   S707_WELD_BUFF_DATA8.RBT7_BT_CODE_NO := W#16#0;
   S707_WELD_BUFF_DATA8.RBT7_WELD_COUNT := W#16#0;
   S707_WELD_BUFF_DATA8.RBT8_BT_CODE_NO := W#16#0;
   S707_WELD_BUFF_DATA8.RBT8_WELD_COUNT := W#16#0;
   S707_WELD_BUFF_DATA8.RBT9_BT_CODE_NO := W#16#0;
   S707_WELD_BUFF_DATA8.RBT9_WELD_COUNT := W#16#0;
   S707_WELD_BUFF_DATA8.RBT10_BT_CODE_NO := W#16#0;
   S707_WELD_BUFF_DATA8.RBT10_WELD_COUNT := W#16#0;
   S707_WELD_BUFF_DATA8.RBT11_BT_CODE_NO := W#16#0;
   S707_WELD_BUFF_DATA8.RBT11_WELD_COUNT := W#16#0;
   S707_WELD_BUFF_DATA8.RBT12_BT_CODE_NO := W#16#0;
   S707_WELD_BUFF_DATA8.RBT12_WELD_COUNT := W#16#0;
   S707_WELD_BUFF_DATA8.RBT13_BT_CODE_NO := W#16#0;
   S707_WELD_BUFF_DATA8.RBT13_WELD_COUNT := W#16#0;
   S707_WELD_BUFF_DATA8.RBT14_BT_CODE_NO := W#16#0;
   S707_WELD_BUFF_DATA8.RBT14_WELD_COUNT := W#16#0;
   S707_WELD_BUFF_DATA8.RBT15_BT_CODE_NO := W#16#0;
   S707_WELD_BUFF_DATA8.RBT15_WELD_COUNT := W#16#0;
   S707_WELD_BUFF_DATA8.RBT16_BT_CODE_NO := W#16#0;
   S707_WELD_BUFF_DATA8.RBT16_WELD_COUNT := W#16#0;
   S707_WELD_BUFF_DATA8.RBT17_BT_CODE_NO := W#16#0;
   S707_WELD_BUFF_DATA8.RBT17_WELD_COUNT := W#16#0;
   S707_WELD_BUFF_DATA8.RBT18_BT_CODE_NO := W#16#0;
   S707_WELD_BUFF_DATA8.RBT18_WELD_COUNT := W#16#0;
   S707_WELD_BUFF_DATA8.RBT19_BT_CODE_NO := W#16#0;
   S707_WELD_BUFF_DATA8.RBT19_WELD_COUNT := W#16#0;
   S707_WELD_BUFF_DATA8.RBT20_BT_CODE_NO := W#16#0;
   S707_WELD_BUFF_DATA8.RBT20_WELD_COUNT := W#16#0;
   S707_WELD_BUFF_DATA8.RBT21_BT_CODE_NO := W#16#0;
   S707_WELD_BUFF_DATA8.RBT21_WELD_COUNT := W#16#0;
   S707_WELD_BUFF_DATA8.RBT22_BT_CODE_NO := W#16#0;
   S707_WELD_BUFF_DATA8.RBT22_WELD_COUNT := W#16#0;
   S707_WELD_BUFF_DATA8.RBT23_BT_CODE_NO := W#16#0;
   S707_WELD_BUFF_DATA8.RBT23_WELD_COUNT := W#16#0;
   S707_WELD_BUFF_DATA8.RBT24_BT_CODE_NO := W#16#0;
   S707_WELD_BUFF_DATA8.RBT24_WELD_COUNT := W#16#0;
   S707_WELD_BUFF_DATA8.WELD_DETERMINES_RESULT := W#16#1;
   S707_WELD_BUFF_DATA8.WELD_CHECK_SUM := W#16#3E;
   S707_WELD_BUFF_DATA8.SPARE1 := W#16#0;
   S707_WELD_BUFF_DATA9.STATION_MAIN := W#16#2C3;
   S707_WELD_BUFF_DATA9.DISTINCTION_LH_RH := W#16#1;
   S707_WELD_BUFF_DATA9.STAION_NUMBER := W#16#0;
   S707_WELD_BUFF_DATA9.VIN_NUMBER1 := W#16#0;
   S707_WELD_BUFF_DATA9.VIN_NUMBER2 := W#16#0;
   S707_WELD_BUFF_DATA9.VIN_NUMBER3 := W#16#0;
   S707_WELD_BUFF_DATA9.VIN_NUMBER4 := W#16#2;
   S707_WELD_BUFF_DATA9.SEQ_NUMBER1 := W#16#14;
   S707_WELD_BUFF_DATA9.SEQ_NUMBER2 := W#16#1795;
   S707_WELD_BUFF_DATA9.RBT1_BT_CODE_NO := W#16#835;
   S707_WELD_BUFF_DATA9.RBT1_WELD_COUNT := W#16#F;
   S707_WELD_BUFF_DATA9.RBT2_BT_CODE_NO := W#16#835;
   S707_WELD_BUFF_DATA9.RBT2_WELD_COUNT := W#16#F;
   S707_WELD_BUFF_DATA9.RBT3_BT_CODE_NO := W#16#835;
   S707_WELD_BUFF_DATA9.RBT3_WELD_COUNT := W#16#11;
   S707_WELD_BUFF_DATA9.RBT4_BT_CODE_NO := W#16#835;
   S707_WELD_BUFF_DATA9.RBT4_WELD_COUNT := W#16#F;
   S707_WELD_BUFF_DATA9.RBT5_BT_CODE_NO := W#16#0;
   S707_WELD_BUFF_DATA9.RBT5_WELD_COUNT := W#16#0;
   S707_WELD_BUFF_DATA9.RBT6_BT_CODE_NO := W#16#0;
   S707_WELD_BUFF_DATA9.RBT6_WELD_COUNT := W#16#0;
   S707_WELD_BUFF_DATA9.RBT7_BT_CODE_NO := W#16#0;
   S707_WELD_BUFF_DATA9.RBT7_WELD_COUNT := W#16#0;
   S707_WELD_BUFF_DATA9.RBT8_BT_CODE_NO := W#16#0;
   S707_WELD_BUFF_DATA9.RBT8_WELD_COUNT := W#16#0;
   S707_WELD_BUFF_DATA9.RBT9_BT_CODE_NO := W#16#0;
   S707_WELD_BUFF_DATA9.RBT9_WELD_COUNT := W#16#0;
   S707_WELD_BUFF_DATA9.RBT10_BT_CODE_NO := W#16#0;
   S707_WELD_BUFF_DATA9.RBT10_WELD_COUNT := W#16#0;
   S707_WELD_BUFF_DATA9.RBT11_BT_CODE_NO := W#16#0;
   S707_WELD_BUFF_DATA9.RBT11_WELD_COUNT := W#16#0;
   S707_WELD_BUFF_DATA9.RBT12_BT_CODE_NO := W#16#0;
   S707_WELD_BUFF_DATA9.RBT12_WELD_COUNT := W#16#0;
   S707_WELD_BUFF_DATA9.RBT13_BT_CODE_NO := W#16#0;
   S707_WELD_BUFF_DATA9.RBT13_WELD_COUNT := W#16#0;
   S707_WELD_BUFF_DATA9.RBT14_BT_CODE_NO := W#16#0;
   S707_WELD_BUFF_DATA9.RBT14_WELD_COUNT := W#16#0;
   S707_WELD_BUFF_DATA9.RBT15_BT_CODE_NO := W#16#0;
   S707_WELD_BUFF_DATA9.RBT15_WELD_COUNT := W#16#0;
   S707_WELD_BUFF_DATA9.RBT16_BT_CODE_NO := W#16#0;
   S707_WELD_BUFF_DATA9.RBT16_WELD_COUNT := W#16#0;
   S707_WELD_BUFF_DATA9.RBT17_BT_CODE_NO := W#16#0;
   S707_WELD_BUFF_DATA9.RBT17_WELD_COUNT := W#16#0;
   S707_WELD_BUFF_DATA9.RBT18_BT_CODE_NO := W#16#0;
   S707_WELD_BUFF_DATA9.RBT18_WELD_COUNT := W#16#0;
   S707_WELD_BUFF_DATA9.RBT19_BT_CODE_NO := W#16#0;
   S707_WELD_BUFF_DATA9.RBT19_WELD_COUNT := W#16#0;
   S707_WELD_BUFF_DATA9.RBT20_BT_CODE_NO := W#16#0;
   S707_WELD_BUFF_DATA9.RBT20_WELD_COUNT := W#16#0;
   S707_WELD_BUFF_DATA9.RBT21_BT_CODE_NO := W#16#0;
   S707_WELD_BUFF_DATA9.RBT21_WELD_COUNT := W#16#0;
   S707_WELD_BUFF_DATA9.RBT22_BT_CODE_NO := W#16#0;
   S707_WELD_BUFF_DATA9.RBT22_WELD_COUNT := W#16#0;
   S707_WELD_BUFF_DATA9.RBT23_BT_CODE_NO := W#16#0;
   S707_WELD_BUFF_DATA9.RBT23_WELD_COUNT := W#16#0;
   S707_WELD_BUFF_DATA9.RBT24_BT_CODE_NO := W#16#0;
   S707_WELD_BUFF_DATA9.RBT24_WELD_COUNT := W#16#0;
   S707_WELD_BUFF_DATA9.WELD_DETERMINES_RESULT := W#16#1;
   S707_WELD_BUFF_DATA9.WELD_CHECK_SUM := W#16#3E;
   S707_WELD_BUFF_DATA9.SPARE1 := W#16#0;
   S707_WELD_BUFF_DATA10.STATION_MAIN := W#16#2C3;
   S707_WELD_BUFF_DATA10.DISTINCTION_LH_RH := W#16#1;
   S707_WELD_BUFF_DATA10.STAION_NUMBER := W#16#0;
   S707_WELD_BUFF_DATA10.VIN_NUMBER1 := W#16#0;
   S707_WELD_BUFF_DATA10.VIN_NUMBER2 := W#16#0;
   S707_WELD_BUFF_DATA10.VIN_NUMBER3 := W#16#0;
   S707_WELD_BUFF_DATA10.VIN_NUMBER4 := W#16#2;
   S707_WELD_BUFF_DATA10.SEQ_NUMBER1 := W#16#14;
   S707_WELD_BUFF_DATA10.SEQ_NUMBER2 := W#16#1794;
   S707_WELD_BUFF_DATA10.RBT1_BT_CODE_NO := W#16#835;
   S707_WELD_BUFF_DATA10.RBT1_WELD_COUNT := W#16#F;
   S707_WELD_BUFF_DATA10.RBT2_BT_CODE_NO := W#16#835;
   S707_WELD_BUFF_DATA10.RBT2_WELD_COUNT := W#16#F;
   S707_WELD_BUFF_DATA10.RBT3_BT_CODE_NO := W#16#835;
   S707_WELD_BUFF_DATA10.RBT3_WELD_COUNT := W#16#11;
   S707_WELD_BUFF_DATA10.RBT4_BT_CODE_NO := W#16#835;
   S707_WELD_BUFF_DATA10.RBT4_WELD_COUNT := W#16#F;
   S707_WELD_BUFF_DATA10.RBT5_BT_CODE_NO := W#16#0;
   S707_WELD_BUFF_DATA10.RBT5_WELD_COUNT := W#16#0;
   S707_WELD_BUFF_DATA10.RBT6_BT_CODE_NO := W#16#0;
   S707_WELD_BUFF_DATA10.RBT6_WELD_COUNT := W#16#0;
   S707_WELD_BUFF_DATA10.RBT7_BT_CODE_NO := W#16#0;
   S707_WELD_BUFF_DATA10.RBT7_WELD_COUNT := W#16#0;
   S707_WELD_BUFF_DATA10.RBT8_BT_CODE_NO := W#16#0;
   S707_WELD_BUFF_DATA10.RBT8_WELD_COUNT := W#16#0;
   S707_WELD_BUFF_DATA10.RBT9_BT_CODE_NO := W#16#0;
   S707_WELD_BUFF_DATA10.RBT9_WELD_COUNT := W#16#0;
   S707_WELD_BUFF_DATA10.RBT10_BT_CODE_NO := W#16#0;
   S707_WELD_BUFF_DATA10.RBT10_WELD_COUNT := W#16#0;
   S707_WELD_BUFF_DATA10.RBT11_BT_CODE_NO := W#16#0;
   S707_WELD_BUFF_DATA10.RBT11_WELD_COUNT := W#16#0;
   S707_WELD_BUFF_DATA10.RBT12_BT_CODE_NO := W#16#0;
   S707_WELD_BUFF_DATA10.RBT12_WELD_COUNT := W#16#0;
   S707_WELD_BUFF_DATA10.RBT13_BT_CODE_NO := W#16#0;
   S707_WELD_BUFF_DATA10.RBT13_WELD_COUNT := W#16#0;
   S707_WELD_BUFF_DATA10.RBT14_BT_CODE_NO := W#16#0;
   S707_WELD_BUFF_DATA10.RBT14_WELD_COUNT := W#16#0;
   S707_WELD_BUFF_DATA10.RBT15_BT_CODE_NO := W#16#0;
   S707_WELD_BUFF_DATA10.RBT15_WELD_COUNT := W#16#0;
   S707_WELD_BUFF_DATA10.RBT16_BT_CODE_NO := W#16#0;
   S707_WELD_BUFF_DATA10.RBT16_WELD_COUNT := W#16#0;
   S707_WELD_BUFF_DATA10.RBT17_BT_CODE_NO := W#16#0;
   S707_WELD_BUFF_DATA10.RBT17_WELD_COUNT := W#16#0;
   S707_WELD_BUFF_DATA10.RBT18_BT_CODE_NO := W#16#0;
   S707_WELD_BUFF_DATA10.RBT18_WELD_COUNT := W#16#0;
   S707_WELD_BUFF_DATA10.RBT19_BT_CODE_NO := W#16#0;
   S707_WELD_BUFF_DATA10.RBT19_WELD_COUNT := W#16#0;
   S707_WELD_BUFF_DATA10.RBT20_BT_CODE_NO := W#16#0;
   S707_WELD_BUFF_DATA10.RBT20_WELD_COUNT := W#16#0;
   S707_WELD_BUFF_DATA10.RBT21_BT_CODE_NO := W#16#0;
   S707_WELD_BUFF_DATA10.RBT21_WELD_COUNT := W#16#0;
   S707_WELD_BUFF_DATA10.RBT22_BT_CODE_NO := W#16#0;
   S707_WELD_BUFF_DATA10.RBT22_WELD_COUNT := W#16#0;
   S707_WELD_BUFF_DATA10.RBT23_BT_CODE_NO := W#16#0;
   S707_WELD_BUFF_DATA10.RBT23_WELD_COUNT := W#16#0;
   S707_WELD_BUFF_DATA10.RBT24_BT_CODE_NO := W#16#0;
   S707_WELD_BUFF_DATA10.RBT24_WELD_COUNT := W#16#0;
   S707_WELD_BUFF_DATA10.WELD_DETERMINES_RESULT := W#16#1;
   S707_WELD_BUFF_DATA10.WELD_CHECK_SUM := W#16#3E;
   S707_WELD_BUFF_DATA10.SPARE1 := W#16#0;
   S707_WELD_BUFF_DATA11.STATION_MAIN := W#16#0;
   S707_WELD_BUFF_DATA11.DISTINCTION_LH_RH := W#16#0;
   S707_WELD_BUFF_DATA11.STAION_NUMBER := W#16#0;
   S707_WELD_BUFF_DATA11.VIN_NUMBER1 := W#16#0;
   S707_WELD_BUFF_DATA11.VIN_NUMBER2 := W#16#0;
   S707_WELD_BUFF_DATA11.VIN_NUMBER3 := W#16#0;
   S707_WELD_BUFF_DATA11.VIN_NUMBER4 := W#16#0;
   S707_WELD_BUFF_DATA11.SEQ_NUMBER1 := W#16#0;
   S707_WELD_BUFF_DATA11.SEQ_NUMBER2 := W#16#0;
   S707_WELD_BUFF_DATA11.RBT1_BT_CODE_NO := W#16#0;
   S707_WELD_BUFF_DATA11.RBT1_WELD_COUNT := W#16#0;
   S707_WELD_BUFF_DATA11.RBT2_BT_CODE_NO := W#16#0;
   S707_WELD_BUFF_DATA11.RBT2_WELD_COUNT := W#16#0;
   S707_WELD_BUFF_DATA11.RBT3_BT_CODE_NO := W#16#0;
   S707_WELD_BUFF_DATA11.RBT3_WELD_COUNT := W#16#0;
   S707_WELD_BUFF_DATA11.RBT4_BT_CODE_NO := W#16#0;
   S707_WELD_BUFF_DATA11.RBT4_WELD_COUNT := W#16#0;
   S707_WELD_BUFF_DATA11.RBT5_BT_CODE_NO := W#16#0;
   S707_WELD_BUFF_DATA11.RBT5_WELD_COUNT := W#16#0;
   S707_WELD_BUFF_DATA11.RBT6_BT_CODE_NO := W#16#0;
   S707_WELD_BUFF_DATA11.RBT6_WELD_COUNT := W#16#0;
   S707_WELD_BUFF_DATA11.RBT7_BT_CODE_NO := W#16#0;
   S707_WELD_BUFF_DATA11.RBT7_WELD_COUNT := W#16#0;
   S707_WELD_BUFF_DATA11.RBT8_BT_CODE_NO := W#16#0;
   S707_WELD_BUFF_DATA11.RBT8_WELD_COUNT := W#16#0;
   S707_WELD_BUFF_DATA11.RBT9_BT_CODE_NO := W#16#0;
   S707_WELD_BUFF_DATA11.RBT9_WELD_COUNT := W#16#0;
   S707_WELD_BUFF_DATA11.RBT10_BT_CODE_NO := W#16#0;
   S707_WELD_BUFF_DATA11.RBT10_WELD_COUNT := W#16#0;
   S707_WELD_BUFF_DATA11.RBT11_BT_CODE_NO := W#16#0;
   S707_WELD_BUFF_DATA11.RBT11_WELD_COUNT := W#16#0;
   S707_WELD_BUFF_DATA11.RBT12_BT_CODE_NO := W#16#0;
   S707_WELD_BUFF_DATA11.RBT12_WELD_COUNT := W#16#0;
   S707_WELD_BUFF_DATA11.RBT13_BT_CODE_NO := W#16#0;
   S707_WELD_BUFF_DATA11.RBT13_WELD_COUNT := W#16#0;
   S707_WELD_BUFF_DATA11.RBT14_BT_CODE_NO := W#16#0;
   S707_WELD_BUFF_DATA11.RBT14_WELD_COUNT := W#16#0;
   S707_WELD_BUFF_DATA11.RBT15_BT_CODE_NO := W#16#0;
   S707_WELD_BUFF_DATA11.RBT15_WELD_COUNT := W#16#0;
   S707_WELD_BUFF_DATA11.RBT16_BT_CODE_NO := W#16#0;
   S707_WELD_BUFF_DATA11.RBT16_WELD_COUNT := W#16#0;
   S707_WELD_BUFF_DATA11.RBT17_BT_CODE_NO := W#16#0;
   S707_WELD_BUFF_DATA11.RBT17_WELD_COUNT := W#16#0;
   S707_WELD_BUFF_DATA11.RBT18_BT_CODE_NO := W#16#0;
   S707_WELD_BUFF_DATA11.RBT18_WELD_COUNT := W#16#0;
   S707_WELD_BUFF_DATA11.RBT19_BT_CODE_NO := W#16#0;
   S707_WELD_BUFF_DATA11.RBT19_WELD_COUNT := W#16#0;
   S707_WELD_BUFF_DATA11.RBT20_BT_CODE_NO := W#16#0;
   S707_WELD_BUFF_DATA11.RBT20_WELD_COUNT := W#16#0;
   S707_WELD_BUFF_DATA11.RBT21_BT_CODE_NO := W#16#0;
   S707_WELD_BUFF_DATA11.RBT21_WELD_COUNT := W#16#0;
   S707_WELD_BUFF_DATA11.RBT22_BT_CODE_NO := W#16#0;
   S707_WELD_BUFF_DATA11.RBT22_WELD_COUNT := W#16#0;
   S707_WELD_BUFF_DATA11.RBT23_BT_CODE_NO := W#16#0;
   S707_WELD_BUFF_DATA11.RBT23_WELD_COUNT := W#16#0;
   S707_WELD_BUFF_DATA11.RBT24_BT_CODE_NO := W#16#0;
   S707_WELD_BUFF_DATA11.RBT24_WELD_COUNT := W#16#0;
   S707_WELD_BUFF_DATA11.WELD_DETERMINES_RESULT := W#16#0;
   S707_WELD_BUFF_DATA11.WELD_CHECK_SUM := W#16#0;
   S707_WELD_BUFF_DATA11.SPARE1 := W#16#0;
   S707_WELD_BUFF_DATA21.STATION_MAIN := W#16#0;
   S707_WELD_BUFF_DATA21.DISTINCTION_LH_RH := W#16#0;
   S707_WELD_BUFF_DATA21.STAION_NUMBER := W#16#0;
   S707_WELD_BUFF_DATA21.VIN_NUMBER1 := W#16#0;
   S707_WELD_BUFF_DATA21.VIN_NUMBER2 := W#16#0;
   S707_WELD_BUFF_DATA21.VIN_NUMBER3 := W#16#0;
   S707_WELD_BUFF_DATA21.VIN_NUMBER4 := W#16#0;
   S707_WELD_BUFF_DATA21.SEQ_NUMBER1 := W#16#0;
   S707_WELD_BUFF_DATA21.SEQ_NUMBER2 := W#16#0;
   S707_WELD_BUFF_DATA21.RBT1_BT_CODE_NO := W#16#0;
   S707_WELD_BUFF_DATA21.RBT1_WELD_COUNT := W#16#0;
   S707_WELD_BUFF_DATA21.RBT2_BT_CODE_NO := W#16#0;
   S707_WELD_BUFF_DATA21.RBT2_WELD_COUNT := W#16#0;
   S707_WELD_BUFF_DATA21.RBT3_BT_CODE_NO := W#16#0;
   S707_WELD_BUFF_DATA21.RBT3_WELD_COUNT := W#16#0;
   S707_WELD_BUFF_DATA21.RBT4_BT_CODE_NO := W#16#0;
   S707_WELD_BUFF_DATA21.RBT4_WELD_COUNT := W#16#0;
   S707_WELD_BUFF_DATA21.RBT5_BT_CODE_NO := W#16#0;
   S707_WELD_BUFF_DATA21.RBT5_WELD_COUNT := W#16#0;
   S707_WELD_BUFF_DATA21.RBT6_BT_CODE_NO := W#16#0;
   S707_WELD_BUFF_DATA21.RBT6_WELD_COUNT := W#16#0;
   S707_WELD_BUFF_DATA21.RBT7_BT_CODE_NO := W#16#0;
   S707_WELD_BUFF_DATA21.RBT7_WELD_COUNT := W#16#0;
   S707_WELD_BUFF_DATA21.RBT8_BT_CODE_NO := W#16#0;
   S707_WELD_BUFF_DATA21.RBT8_WELD_COUNT := W#16#0;
   S707_WELD_BUFF_DATA21.RBT9_BT_CODE_NO := W#16#0;
   S707_WELD_BUFF_DATA21.RBT9_WELD_COUNT := W#16#0;
   S707_WELD_BUFF_DATA21.RBT10_BT_CODE_NO := W#16#0;
   S707_WELD_BUFF_DATA21.RBT10_WELD_COUNT := W#16#0;
   S707_WELD_BUFF_DATA21.RBT11_BT_CODE_NO := W#16#0;
   S707_WELD_BUFF_DATA21.RBT11_WELD_COUNT := W#16#0;
   S707_WELD_BUFF_DATA21.RBT12_BT_CODE_NO := W#16#0;
   S707_WELD_BUFF_DATA21.RBT12_WELD_COUNT := W#16#0;
   S707_WELD_BUFF_DATA21.RBT13_BT_CODE_NO := W#16#0;
   S707_WELD_BUFF_DATA21.RBT13_WELD_COUNT := W#16#0;
   S707_WELD_BUFF_DATA21.RBT14_BT_CODE_NO := W#16#0;
   S707_WELD_BUFF_DATA21.RBT14_WELD_COUNT := W#16#0;
   S707_WELD_BUFF_DATA21.RBT15_BT_CODE_NO := W#16#0;
   S707_WELD_BUFF_DATA21.RBT15_WELD_COUNT := W#16#0;
   S707_WELD_BUFF_DATA21.RBT16_BT_CODE_NO := W#16#0;
   S707_WELD_BUFF_DATA21.RBT16_WELD_COUNT := W#16#0;
   S707_WELD_BUFF_DATA21.RBT17_BT_CODE_NO := W#16#0;
   S707_WELD_BUFF_DATA21.RBT17_WELD_COUNT := W#16#0;
   S707_WELD_BUFF_DATA21.RBT18_BT_CODE_NO := W#16#0;
   S707_WELD_BUFF_DATA21.RBT18_WELD_COUNT := W#16#0;
   S707_WELD_BUFF_DATA21.RBT19_BT_CODE_NO := W#16#0;
   S707_WELD_BUFF_DATA21.RBT19_WELD_COUNT := W#16#0;
   S707_WELD_BUFF_DATA21.RBT20_BT_CODE_NO := W#16#0;
   S707_WELD_BUFF_DATA21.RBT20_WELD_COUNT := W#16#0;
   S707_WELD_BUFF_DATA21.RBT21_BT_CODE_NO := W#16#0;
   S707_WELD_BUFF_DATA21.RBT21_WELD_COUNT := W#16#0;
   S707_WELD_BUFF_DATA21.RBT22_BT_CODE_NO := W#16#0;
   S707_WELD_BUFF_DATA21.RBT22_WELD_COUNT := W#16#0;
   S707_WELD_BUFF_DATA21.RBT23_BT_CODE_NO := W#16#0;
   S707_WELD_BUFF_DATA21.RBT23_WELD_COUNT := W#16#0;
   S707_WELD_BUFF_DATA21.RBT24_BT_CODE_NO := W#16#0;
   S707_WELD_BUFF_DATA21.RBT24_WELD_COUNT := W#16#0;
   S707_WELD_BUFF_DATA21.WELD_DETERMINES_RESULT := W#16#0;
   S707_WELD_BUFF_DATA21.WELD_CHECK_SUM := W#16#0;
   S707_WELD_BUFF_DATA21.SPARE1 := W#16#0;
   S707_WELD_BUFF_DATA31.STATION_MAIN := W#16#0;
   S707_WELD_BUFF_DATA31.DISTINCTION_LH_RH := W#16#0;
   S707_WELD_BUFF_DATA31.STAION_NUMBER := W#16#0;
   S707_WELD_BUFF_DATA31.VIN_NUMBER1 := W#16#0;
   S707_WELD_BUFF_DATA31.VIN_NUMBER2 := W#16#0;
   S707_WELD_BUFF_DATA31.VIN_NUMBER3 := W#16#0;
   S707_WELD_BUFF_DATA31.VIN_NUMBER4 := W#16#0;
   S707_WELD_BUFF_DATA31.SEQ_NUMBER1 := W#16#0;
   S707_WELD_BUFF_DATA31.SEQ_NUMBER2 := W#16#0;
   S707_WELD_BUFF_DATA31.RBT1_BT_CODE_NO := W#16#0;
   S707_WELD_BUFF_DATA31.RBT1_WELD_COUNT := W#16#0;
   S707_WELD_BUFF_DATA31.RBT2_BT_CODE_NO := W#16#0;
   S707_WELD_BUFF_DATA31.RBT2_WELD_COUNT := W#16#0;
   S707_WELD_BUFF_DATA31.RBT3_BT_CODE_NO := W#16#0;
   S707_WELD_BUFF_DATA31.RBT3_WELD_COUNT := W#16#0;
   S707_WELD_BUFF_DATA31.RBT4_BT_CODE_NO := W#16#0;
   S707_WELD_BUFF_DATA31.RBT4_WELD_COUNT := W#16#0;
   S707_WELD_BUFF_DATA31.RBT5_BT_CODE_NO := W#16#0;
   S707_WELD_BUFF_DATA31.RBT5_WELD_COUNT := W#16#0;
   S707_WELD_BUFF_DATA31.RBT6_BT_CODE_NO := W#16#0;
   S707_WELD_BUFF_DATA31.RBT6_WELD_COUNT := W#16#0;
   S707_WELD_BUFF_DATA31.RBT7_BT_CODE_NO := W#16#0;
   S707_WELD_BUFF_DATA31.RBT7_WELD_COUNT := W#16#0;
   S707_WELD_BUFF_DATA31.RBT8_BT_CODE_NO := W#16#0;
   S707_WELD_BUFF_DATA31.RBT8_WELD_COUNT := W#16#0;
   S707_WELD_BUFF_DATA31.RBT9_BT_CODE_NO := W#16#0;
   S707_WELD_BUFF_DATA31.RBT9_WELD_COUNT := W#16#0;
   S707_WELD_BUFF_DATA31.RBT10_BT_CODE_NO := W#16#0;
   S707_WELD_BUFF_DATA31.RBT10_WELD_COUNT := W#16#0;
   S707_WELD_BUFF_DATA31.RBT11_BT_CODE_NO := W#16#0;
   S707_WELD_BUFF_DATA31.RBT11_WELD_COUNT := W#16#0;
   S707_WELD_BUFF_DATA31.RBT12_BT_CODE_NO := W#16#0;
   S707_WELD_BUFF_DATA31.RBT12_WELD_COUNT := W#16#0;
   S707_WELD_BUFF_DATA31.RBT13_BT_CODE_NO := W#16#0;
   S707_WELD_BUFF_DATA31.RBT13_WELD_COUNT := W#16#0;
   S707_WELD_BUFF_DATA31.RBT14_BT_CODE_NO := W#16#0;
   S707_WELD_BUFF_DATA31.RBT14_WELD_COUNT := W#16#0;
   S707_WELD_BUFF_DATA31.RBT15_BT_CODE_NO := W#16#0;
   S707_WELD_BUFF_DATA31.RBT15_WELD_COUNT := W#16#0;
   S707_WELD_BUFF_DATA31.RBT16_BT_CODE_NO := W#16#0;
   S707_WELD_BUFF_DATA31.RBT16_WELD_COUNT := W#16#0;
   S707_WELD_BUFF_DATA31.RBT17_BT_CODE_NO := W#16#0;
   S707_WELD_BUFF_DATA31.RBT17_WELD_COUNT := W#16#0;
   S707_WELD_BUFF_DATA31.RBT18_BT_CODE_NO := W#16#0;
   S707_WELD_BUFF_DATA31.RBT18_WELD_COUNT := W#16#0;
   S707_WELD_BUFF_DATA31.RBT19_BT_CODE_NO := W#16#0;
   S707_WELD_BUFF_DATA31.RBT19_WELD_COUNT := W#16#0;
   S707_WELD_BUFF_DATA31.RBT20_BT_CODE_NO := W#16#0;
   S707_WELD_BUFF_DATA31.RBT20_WELD_COUNT := W#16#0;
   S707_WELD_BUFF_DATA31.RBT21_BT_CODE_NO := W#16#0;
   S707_WELD_BUFF_DATA31.RBT21_WELD_COUNT := W#16#0;
   S707_WELD_BUFF_DATA31.RBT22_BT_CODE_NO := W#16#0;
   S707_WELD_BUFF_DATA31.RBT22_WELD_COUNT := W#16#0;
   S707_WELD_BUFF_DATA31.RBT23_BT_CODE_NO := W#16#0;
   S707_WELD_BUFF_DATA31.RBT23_WELD_COUNT := W#16#0;
   S707_WELD_BUFF_DATA31.RBT24_BT_CODE_NO := W#16#0;
   S707_WELD_BUFF_DATA31.RBT24_WELD_COUNT := W#16#0;
   S707_WELD_BUFF_DATA31.WELD_DETERMINES_RESULT := W#16#0;
   S707_WELD_BUFF_DATA31.WELD_CHECK_SUM := W#16#0;
   S707_WELD_BUFF_DATA31.SPARE1 := W#16#0;
   S707_WELD_BUFF_DATA41.STATION_MAIN := W#16#0;
   S707_WELD_BUFF_DATA41.DISTINCTION_LH_RH := W#16#0;
   S707_WELD_BUFF_DATA41.STAION_NUMBER := W#16#0;
   S707_WELD_BUFF_DATA41.VIN_NUMBER1 := W#16#0;
   S707_WELD_BUFF_DATA41.VIN_NUMBER2 := W#16#0;
   S707_WELD_BUFF_DATA41.VIN_NUMBER3 := W#16#0;
   S707_WELD_BUFF_DATA41.VIN_NUMBER4 := W#16#0;
   S707_WELD_BUFF_DATA41.SEQ_NUMBER1 := W#16#0;
   S707_WELD_BUFF_DATA41.SEQ_NUMBER2 := W#16#0;
   S707_WELD_BUFF_DATA41.RBT1_BT_CODE_NO := W#16#0;
   S707_WELD_BUFF_DATA41.RBT1_WELD_COUNT := W#16#0;
   S707_WELD_BUFF_DATA41.RBT2_BT_CODE_NO := W#16#0;
   S707_WELD_BUFF_DATA41.RBT2_WELD_COUNT := W#16#0;
   S707_WELD_BUFF_DATA41.RBT3_BT_CODE_NO := W#16#0;
   S707_WELD_BUFF_DATA41.RBT3_WELD_COUNT := W#16#0;
   S707_WELD_BUFF_DATA41.RBT4_BT_CODE_NO := W#16#0;
   S707_WELD_BUFF_DATA41.RBT4_WELD_COUNT := W#16#0;
   S707_WELD_BUFF_DATA41.RBT5_BT_CODE_NO := W#16#0;
   S707_WELD_BUFF_DATA41.RBT5_WELD_COUNT := W#16#0;
   S707_WELD_BUFF_DATA41.RBT6_BT_CODE_NO := W#16#0;
   S707_WELD_BUFF_DATA41.RBT6_WELD_COUNT := W#16#0;
   S707_WELD_BUFF_DATA41.RBT7_BT_CODE_NO := W#16#0;
   S707_WELD_BUFF_DATA41.RBT7_WELD_COUNT := W#16#0;
   S707_WELD_BUFF_DATA41.RBT8_BT_CODE_NO := W#16#0;
   S707_WELD_BUFF_DATA41.RBT8_WELD_COUNT := W#16#0;
   S707_WELD_BUFF_DATA41.RBT9_BT_CODE_NO := W#16#0;
   S707_WELD_BUFF_DATA41.RBT9_WELD_COUNT := W#16#0;
   S707_WELD_BUFF_DATA41.RBT10_BT_CODE_NO := W#16#0;
   S707_WELD_BUFF_DATA41.RBT10_WELD_COUNT := W#16#0;
   S707_WELD_BUFF_DATA41.RBT11_BT_CODE_NO := W#16#0;
   S707_WELD_BUFF_DATA41.RBT11_WELD_COUNT := W#16#0;
   S707_WELD_BUFF_DATA41.RBT12_BT_CODE_NO := W#16#0;
   S707_WELD_BUFF_DATA41.RBT12_WELD_COUNT := W#16#0;
   S707_WELD_BUFF_DATA41.RBT13_BT_CODE_NO := W#16#0;
   S707_WELD_BUFF_DATA41.RBT13_WELD_COUNT := W#16#0;
   S707_WELD_BUFF_DATA41.RBT14_BT_CODE_NO := W#16#0;
   S707_WELD_BUFF_DATA41.RBT14_WELD_COUNT := W#16#0;
   S707_WELD_BUFF_DATA41.RBT15_BT_CODE_NO := W#16#0;
   S707_WELD_BUFF_DATA41.RBT15_WELD_COUNT := W#16#0;
   S707_WELD_BUFF_DATA41.RBT16_BT_CODE_NO := W#16#0;
   S707_WELD_BUFF_DATA41.RBT16_WELD_COUNT := W#16#0;
   S707_WELD_BUFF_DATA41.RBT17_BT_CODE_NO := W#16#0;
   S707_WELD_BUFF_DATA41.RBT17_WELD_COUNT := W#16#0;
   S707_WELD_BUFF_DATA41.RBT18_BT_CODE_NO := W#16#0;
   S707_WELD_BUFF_DATA41.RBT18_WELD_COUNT := W#16#0;
   S707_WELD_BUFF_DATA41.RBT19_BT_CODE_NO := W#16#0;
   S707_WELD_BUFF_DATA41.RBT19_WELD_COUNT := W#16#0;
   S707_WELD_BUFF_DATA41.RBT20_BT_CODE_NO := W#16#0;
   S707_WELD_BUFF_DATA41.RBT20_WELD_COUNT := W#16#0;
   S707_WELD_BUFF_DATA41.RBT21_BT_CODE_NO := W#16#0;
   S707_WELD_BUFF_DATA41.RBT21_WELD_COUNT := W#16#0;
   S707_WELD_BUFF_DATA41.RBT22_BT_CODE_NO := W#16#0;
   S707_WELD_BUFF_DATA41.RBT22_WELD_COUNT := W#16#0;
   S707_WELD_BUFF_DATA41.RBT23_BT_CODE_NO := W#16#0;
   S707_WELD_BUFF_DATA41.RBT23_WELD_COUNT := W#16#0;
   S707_WELD_BUFF_DATA41.RBT24_BT_CODE_NO := W#16#0;
   S707_WELD_BUFF_DATA41.RBT24_WELD_COUNT := W#16#0;
   S707_WELD_BUFF_DATA41.WELD_DETERMINES_RESULT := W#16#0;
   S707_WELD_BUFF_DATA41.WELD_CHECK_SUM := W#16#0;
   S707_WELD_BUFF_DATA41.SPARE1 := W#16#0;
   S707_WELD_BUFF_DATA51.STATION_MAIN := W#16#0;
   S707_WELD_BUFF_DATA51.DISTINCTION_LH_RH := W#16#0;
   S707_WELD_BUFF_DATA51.STAION_NUMBER := W#16#0;
   S707_WELD_BUFF_DATA51.VIN_NUMBER1 := W#16#0;
   S707_WELD_BUFF_DATA51.VIN_NUMBER2 := W#16#0;
   S707_WELD_BUFF_DATA51.VIN_NUMBER3 := W#16#0;
   S707_WELD_BUFF_DATA51.VIN_NUMBER4 := W#16#0;
   S707_WELD_BUFF_DATA51.SEQ_NUMBER1 := W#16#0;
   S707_WELD_BUFF_DATA51.SEQ_NUMBER2 := W#16#0;
   S707_WELD_BUFF_DATA51.RBT1_BT_CODE_NO := W#16#0;
   S707_WELD_BUFF_DATA51.RBT1_WELD_COUNT := W#16#0;
   S707_WELD_BUFF_DATA51.RBT2_BT_CODE_NO := W#16#0;
   S707_WELD_BUFF_DATA51.RBT2_WELD_COUNT := W#16#0;
   S707_WELD_BUFF_DATA51.RBT3_BT_CODE_NO := W#16#0;
   S707_WELD_BUFF_DATA51.RBT3_WELD_COUNT := W#16#0;
   S707_WELD_BUFF_DATA51.RBT4_BT_CODE_NO := W#16#0;
   S707_WELD_BUFF_DATA51.RBT4_WELD_COUNT := W#16#0;
   S707_WELD_BUFF_DATA51.RBT5_BT_CODE_NO := W#16#0;
   S707_WELD_BUFF_DATA51.RBT5_WELD_COUNT := W#16#0;
   S707_WELD_BUFF_DATA51.RBT6_BT_CODE_NO := W#16#0;
   S707_WELD_BUFF_DATA51.RBT6_WELD_COUNT := W#16#0;
   S707_WELD_BUFF_DATA51.RBT7_BT_CODE_NO := W#16#0;
   S707_WELD_BUFF_DATA51.RBT7_WELD_COUNT := W#16#0;
   S707_WELD_BUFF_DATA51.RBT8_BT_CODE_NO := W#16#0;
   S707_WELD_BUFF_DATA51.RBT8_WELD_COUNT := W#16#0;
   S707_WELD_BUFF_DATA51.RBT9_BT_CODE_NO := W#16#0;
   S707_WELD_BUFF_DATA51.RBT9_WELD_COUNT := W#16#0;
   S707_WELD_BUFF_DATA51.RBT10_BT_CODE_NO := W#16#0;
   S707_WELD_BUFF_DATA51.RBT10_WELD_COUNT := W#16#0;
   S707_WELD_BUFF_DATA51.RBT11_BT_CODE_NO := W#16#0;
   S707_WELD_BUFF_DATA51.RBT11_WELD_COUNT := W#16#0;
   S707_WELD_BUFF_DATA51.RBT12_BT_CODE_NO := W#16#0;
   S707_WELD_BUFF_DATA51.RBT12_WELD_COUNT := W#16#0;
   S707_WELD_BUFF_DATA51.RBT13_BT_CODE_NO := W#16#0;
   S707_WELD_BUFF_DATA51.RBT13_WELD_COUNT := W#16#0;
   S707_WELD_BUFF_DATA51.RBT14_BT_CODE_NO := W#16#0;
   S707_WELD_BUFF_DATA51.RBT14_WELD_COUNT := W#16#0;
   S707_WELD_BUFF_DATA51.RBT15_BT_CODE_NO := W#16#0;
   S707_WELD_BUFF_DATA51.RBT15_WELD_COUNT := W#16#0;
   S707_WELD_BUFF_DATA51.RBT16_BT_CODE_NO := W#16#0;
   S707_WELD_BUFF_DATA51.RBT16_WELD_COUNT := W#16#0;
   S707_WELD_BUFF_DATA51.RBT17_BT_CODE_NO := W#16#0;
   S707_WELD_BUFF_DATA51.RBT17_WELD_COUNT := W#16#0;
   S707_WELD_BUFF_DATA51.RBT18_BT_CODE_NO := W#16#0;
   S707_WELD_BUFF_DATA51.RBT18_WELD_COUNT := W#16#0;
   S707_WELD_BUFF_DATA51.RBT19_BT_CODE_NO := W#16#0;
   S707_WELD_BUFF_DATA51.RBT19_WELD_COUNT := W#16#0;
   S707_WELD_BUFF_DATA51.RBT20_BT_CODE_NO := W#16#0;
   S707_WELD_BUFF_DATA51.RBT20_WELD_COUNT := W#16#0;
   S707_WELD_BUFF_DATA51.RBT21_BT_CODE_NO := W#16#0;
   S707_WELD_BUFF_DATA51.RBT21_WELD_COUNT := W#16#0;
   S707_WELD_BUFF_DATA51.RBT22_BT_CODE_NO := W#16#0;
   S707_WELD_BUFF_DATA51.RBT22_WELD_COUNT := W#16#0;
   S707_WELD_BUFF_DATA51.RBT23_BT_CODE_NO := W#16#0;
   S707_WELD_BUFF_DATA51.RBT23_WELD_COUNT := W#16#0;
   S707_WELD_BUFF_DATA51.RBT24_BT_CODE_NO := W#16#0;
   S707_WELD_BUFF_DATA51.RBT24_WELD_COUNT := W#16#0;
   S707_WELD_BUFF_DATA51.WELD_DETERMINES_RESULT := W#16#0;
   S707_WELD_BUFF_DATA51.WELD_CHECK_SUM := W#16#0;
   S707_WELD_BUFF_DATA51.SPARE1 := W#16#0;
   S707_WELD_BUFF_DATA61.STATION_MAIN := W#16#0;
   S707_WELD_BUFF_DATA61.DISTINCTION_LH_RH := W#16#0;
   S707_WELD_BUFF_DATA61.STAION_NUMBER := W#16#0;
   S707_WELD_BUFF_DATA61.VIN_NUMBER1 := W#16#0;
   S707_WELD_BUFF_DATA61.VIN_NUMBER2 := W#16#0;
   S707_WELD_BUFF_DATA61.VIN_NUMBER3 := W#16#0;
   S707_WELD_BUFF_DATA61.VIN_NUMBER4 := W#16#0;
   S707_WELD_BUFF_DATA61.SEQ_NUMBER1 := W#16#0;
   S707_WELD_BUFF_DATA61.SEQ_NUMBER2 := W#16#0;
   S707_WELD_BUFF_DATA61.RBT1_BT_CODE_NO := W#16#0;
   S707_WELD_BUFF_DATA61.RBT1_WELD_COUNT := W#16#0;
   S707_WELD_BUFF_DATA61.RBT2_BT_CODE_NO := W#16#0;
   S707_WELD_BUFF_DATA61.RBT2_WELD_COUNT := W#16#0;
   S707_WELD_BUFF_DATA61.RBT3_BT_CODE_NO := W#16#0;
   S707_WELD_BUFF_DATA61.RBT3_WELD_COUNT := W#16#0;
   S707_WELD_BUFF_DATA61.RBT4_BT_CODE_NO := W#16#0;
   S707_WELD_BUFF_DATA61.RBT4_WELD_COUNT := W#16#0;
   S707_WELD_BUFF_DATA61.RBT5_BT_CODE_NO := W#16#0;
   S707_WELD_BUFF_DATA61.RBT5_WELD_COUNT := W#16#0;
   S707_WELD_BUFF_DATA61.RBT6_BT_CODE_NO := W#16#0;
   S707_WELD_BUFF_DATA61.RBT6_WELD_COUNT := W#16#0;
   S707_WELD_BUFF_DATA61.RBT7_BT_CODE_NO := W#16#0;
   S707_WELD_BUFF_DATA61.RBT7_WELD_COUNT := W#16#0;
   S707_WELD_BUFF_DATA61.RBT8_BT_CODE_NO := W#16#0;
   S707_WELD_BUFF_DATA61.RBT8_WELD_COUNT := W#16#0;
   S707_WELD_BUFF_DATA61.RBT9_BT_CODE_NO := W#16#0;
   S707_WELD_BUFF_DATA61.RBT9_WELD_COUNT := W#16#0;
   S707_WELD_BUFF_DATA61.RBT10_BT_CODE_NO := W#16#0;
   S707_WELD_BUFF_DATA61.RBT10_WELD_COUNT := W#16#0;
   S707_WELD_BUFF_DATA61.RBT11_BT_CODE_NO := W#16#0;
   S707_WELD_BUFF_DATA61.RBT11_WELD_COUNT := W#16#0;
   S707_WELD_BUFF_DATA61.RBT12_BT_CODE_NO := W#16#0;
   S707_WELD_BUFF_DATA61.RBT12_WELD_COUNT := W#16#0;
   S707_WELD_BUFF_DATA61.RBT13_BT_CODE_NO := W#16#0;
   S707_WELD_BUFF_DATA61.RBT13_WELD_COUNT := W#16#0;
   S707_WELD_BUFF_DATA61.RBT14_BT_CODE_NO := W#16#0;
   S707_WELD_BUFF_DATA61.RBT14_WELD_COUNT := W#16#0;
   S707_WELD_BUFF_DATA61.RBT15_BT_CODE_NO := W#16#0;
   S707_WELD_BUFF_DATA61.RBT15_WELD_COUNT := W#16#0;
   S707_WELD_BUFF_DATA61.RBT16_BT_CODE_NO := W#16#0;
   S707_WELD_BUFF_DATA61.RBT16_WELD_COUNT := W#16#0;
   S707_WELD_BUFF_DATA61.RBT17_BT_CODE_NO := W#16#0;
   S707_WELD_BUFF_DATA61.RBT17_WELD_COUNT := W#16#0;
   S707_WELD_BUFF_DATA61.RBT18_BT_CODE_NO := W#16#0;
   S707_WELD_BUFF_DATA61.RBT18_WELD_COUNT := W#16#0;
   S707_WELD_BUFF_DATA61.RBT19_BT_CODE_NO := W#16#0;
   S707_WELD_BUFF_DATA61.RBT19_WELD_COUNT := W#16#0;
   S707_WELD_BUFF_DATA61.RBT20_BT_CODE_NO := W#16#0;
   S707_WELD_BUFF_DATA61.RBT20_WELD_COUNT := W#16#0;
   S707_WELD_BUFF_DATA61.RBT21_BT_CODE_NO := W#16#0;
   S707_WELD_BUFF_DATA61.RBT21_WELD_COUNT := W#16#0;
   S707_WELD_BUFF_DATA61.RBT22_BT_CODE_NO := W#16#0;
   S707_WELD_BUFF_DATA61.RBT22_WELD_COUNT := W#16#0;
   S707_WELD_BUFF_DATA61.RBT23_BT_CODE_NO := W#16#0;
   S707_WELD_BUFF_DATA61.RBT23_WELD_COUNT := W#16#0;
   S707_WELD_BUFF_DATA61.RBT24_BT_CODE_NO := W#16#0;
   S707_WELD_BUFF_DATA61.RBT24_WELD_COUNT := W#16#0;
   S707_WELD_BUFF_DATA61.WELD_DETERMINES_RESULT := W#16#0;
   S707_WELD_BUFF_DATA61.WELD_CHECK_SUM := W#16#0;
   S707_WELD_BUFF_DATA61.SPARE1 := W#16#0;
   S707_WELD_BUFF_DATA71.STATION_MAIN := W#16#0;
   S707_WELD_BUFF_DATA71.DISTINCTION_LH_RH := W#16#0;
   S707_WELD_BUFF_DATA71.STAION_NUMBER := W#16#0;
   S707_WELD_BUFF_DATA71.VIN_NUMBER1 := W#16#0;
   S707_WELD_BUFF_DATA71.VIN_NUMBER2 := W#16#0;
   S707_WELD_BUFF_DATA71.VIN_NUMBER3 := W#16#0;
   S707_WELD_BUFF_DATA71.VIN_NUMBER4 := W#16#0;
   S707_WELD_BUFF_DATA71.SEQ_NUMBER1 := W#16#0;
   S707_WELD_BUFF_DATA71.SEQ_NUMBER2 := W#16#0;
   S707_WELD_BUFF_DATA71.RBT1_BT_CODE_NO := W#16#0;
   S707_WELD_BUFF_DATA71.RBT1_WELD_COUNT := W#16#0;
   S707_WELD_BUFF_DATA71.RBT2_BT_CODE_NO := W#16#0;
   S707_WELD_BUFF_DATA71.RBT2_WELD_COUNT := W#16#0;
   S707_WELD_BUFF_DATA71.RBT3_BT_CODE_NO := W#16#0;
   S707_WELD_BUFF_DATA71.RBT3_WELD_COUNT := W#16#0;
   S707_WELD_BUFF_DATA71.RBT4_BT_CODE_NO := W#16#0;
   S707_WELD_BUFF_DATA71.RBT4_WELD_COUNT := W#16#0;
   S707_WELD_BUFF_DATA71.RBT5_BT_CODE_NO := W#16#0;
   S707_WELD_BUFF_DATA71.RBT5_WELD_COUNT := W#16#0;
   S707_WELD_BUFF_DATA71.RBT6_BT_CODE_NO := W#16#0;
   S707_WELD_BUFF_DATA71.RBT6_WELD_COUNT := W#16#0;
   S707_WELD_BUFF_DATA71.RBT7_BT_CODE_NO := W#16#0;
   S707_WELD_BUFF_DATA71.RBT7_WELD_COUNT := W#16#0;
   S707_WELD_BUFF_DATA71.RBT8_BT_CODE_NO := W#16#0;
   S707_WELD_BUFF_DATA71.RBT8_WELD_COUNT := W#16#0;
   S707_WELD_BUFF_DATA71.RBT9_BT_CODE_NO := W#16#0;
   S707_WELD_BUFF_DATA71.RBT9_WELD_COUNT := W#16#0;
   S707_WELD_BUFF_DATA71.RBT10_BT_CODE_NO := W#16#0;
   S707_WELD_BUFF_DATA71.RBT10_WELD_COUNT := W#16#0;
   S707_WELD_BUFF_DATA71.RBT11_BT_CODE_NO := W#16#0;
   S707_WELD_BUFF_DATA71.RBT11_WELD_COUNT := W#16#0;
   S707_WELD_BUFF_DATA71.RBT12_BT_CODE_NO := W#16#0;
   S707_WELD_BUFF_DATA71.RBT12_WELD_COUNT := W#16#0;
   S707_WELD_BUFF_DATA71.RBT13_BT_CODE_NO := W#16#0;
   S707_WELD_BUFF_DATA71.RBT13_WELD_COUNT := W#16#0;
   S707_WELD_BUFF_DATA71.RBT14_BT_CODE_NO := W#16#0;
   S707_WELD_BUFF_DATA71.RBT14_WELD_COUNT := W#16#0;
   S707_WELD_BUFF_DATA71.RBT15_BT_CODE_NO := W#16#0;
   S707_WELD_BUFF_DATA71.RBT15_WELD_COUNT := W#16#0;
   S707_WELD_BUFF_DATA71.RBT16_BT_CODE_NO := W#16#0;
   S707_WELD_BUFF_DATA71.RBT16_WELD_COUNT := W#16#0;
   S707_WELD_BUFF_DATA71.RBT17_BT_CODE_NO := W#16#0;
   S707_WELD_BUFF_DATA71.RBT17_WELD_COUNT := W#16#0;
   S707_WELD_BUFF_DATA71.RBT18_BT_CODE_NO := W#16#0;
   S707_WELD_BUFF_DATA71.RBT18_WELD_COUNT := W#16#0;
   S707_WELD_BUFF_DATA71.RBT19_BT_CODE_NO := W#16#0;
   S707_WELD_BUFF_DATA71.RBT19_WELD_COUNT := W#16#0;
   S707_WELD_BUFF_DATA71.RBT20_BT_CODE_NO := W#16#0;
   S707_WELD_BUFF_DATA71.RBT20_WELD_COUNT := W#16#0;
   S707_WELD_BUFF_DATA71.RBT21_BT_CODE_NO := W#16#0;
   S707_WELD_BUFF_DATA71.RBT21_WELD_COUNT := W#16#0;
   S707_WELD_BUFF_DATA71.RBT22_BT_CODE_NO := W#16#0;
   S707_WELD_BUFF_DATA71.RBT22_WELD_COUNT := W#16#0;
   S707_WELD_BUFF_DATA71.RBT23_BT_CODE_NO := W#16#0;
   S707_WELD_BUFF_DATA71.RBT23_WELD_COUNT := W#16#0;
   S707_WELD_BUFF_DATA71.RBT24_BT_CODE_NO := W#16#0;
   S707_WELD_BUFF_DATA71.RBT24_WELD_COUNT := W#16#0;
   S707_WELD_BUFF_DATA71.WELD_DETERMINES_RESULT := W#16#0;
   S707_WELD_BUFF_DATA71.WELD_CHECK_SUM := W#16#0;
   S707_WELD_BUFF_DATA71.SPARE1 := W#16#0;
   S707_WELD_BUFF_DATA81.STATION_MAIN := W#16#0;
   S707_WELD_BUFF_DATA81.DISTINCTION_LH_RH := W#16#0;
   S707_WELD_BUFF_DATA81.STAION_NUMBER := W#16#0;
   S707_WELD_BUFF_DATA81.VIN_NUMBER1 := W#16#0;
   S707_WELD_BUFF_DATA81.VIN_NUMBER2 := W#16#0;
   S707_WELD_BUFF_DATA81.VIN_NUMBER3 := W#16#0;
   S707_WELD_BUFF_DATA81.VIN_NUMBER4 := W#16#0;
   S707_WELD_BUFF_DATA81.SEQ_NUMBER1 := W#16#0;
   S707_WELD_BUFF_DATA81.SEQ_NUMBER2 := W#16#0;
   S707_WELD_BUFF_DATA81.RBT1_BT_CODE_NO := W#16#0;
   S707_WELD_BUFF_DATA81.RBT1_WELD_COUNT := W#16#0;
   S707_WELD_BUFF_DATA81.RBT2_BT_CODE_NO := W#16#0;
   S707_WELD_BUFF_DATA81.RBT2_WELD_COUNT := W#16#0;
   S707_WELD_BUFF_DATA81.RBT3_BT_CODE_NO := W#16#0;
   S707_WELD_BUFF_DATA81.RBT3_WELD_COUNT := W#16#0;
   S707_WELD_BUFF_DATA81.RBT4_BT_CODE_NO := W#16#0;
   S707_WELD_BUFF_DATA81.RBT4_WELD_COUNT := W#16#0;
   S707_WELD_BUFF_DATA81.RBT5_BT_CODE_NO := W#16#0;
   S707_WELD_BUFF_DATA81.RBT5_WELD_COUNT := W#16#0;
   S707_WELD_BUFF_DATA81.RBT6_BT_CODE_NO := W#16#0;
   S707_WELD_BUFF_DATA81.RBT6_WELD_COUNT := W#16#0;
   S707_WELD_BUFF_DATA81.RBT7_BT_CODE_NO := W#16#0;
   S707_WELD_BUFF_DATA81.RBT7_WELD_COUNT := W#16#0;
   S707_WELD_BUFF_DATA81.RBT8_BT_CODE_NO := W#16#0;
   S707_WELD_BUFF_DATA81.RBT8_WELD_COUNT := W#16#0;
   S707_WELD_BUFF_DATA81.RBT9_BT_CODE_NO := W#16#0;
   S707_WELD_BUFF_DATA81.RBT9_WELD_COUNT := W#16#0;
   S707_WELD_BUFF_DATA81.RBT10_BT_CODE_NO := W#16#0;
   S707_WELD_BUFF_DATA81.RBT10_WELD_COUNT := W#16#0;
   S707_WELD_BUFF_DATA81.RBT11_BT_CODE_NO := W#16#0;
   S707_WELD_BUFF_DATA81.RBT11_WELD_COUNT := W#16#0;
   S707_WELD_BUFF_DATA81.RBT12_BT_CODE_NO := W#16#0;
   S707_WELD_BUFF_DATA81.RBT12_WELD_COUNT := W#16#0;
   S707_WELD_BUFF_DATA81.RBT13_BT_CODE_NO := W#16#0;
   S707_WELD_BUFF_DATA81.RBT13_WELD_COUNT := W#16#0;
   S707_WELD_BUFF_DATA81.RBT14_BT_CODE_NO := W#16#0;
   S707_WELD_BUFF_DATA81.RBT14_WELD_COUNT := W#16#0;
   S707_WELD_BUFF_DATA81.RBT15_BT_CODE_NO := W#16#0;
   S707_WELD_BUFF_DATA81.RBT15_WELD_COUNT := W#16#0;
   S707_WELD_BUFF_DATA81.RBT16_BT_CODE_NO := W#16#0;
   S707_WELD_BUFF_DATA81.RBT16_WELD_COUNT := W#16#0;
   S707_WELD_BUFF_DATA81.RBT17_BT_CODE_NO := W#16#0;
   S707_WELD_BUFF_DATA81.RBT17_WELD_COUNT := W#16#0;
   S707_WELD_BUFF_DATA81.RBT18_BT_CODE_NO := W#16#0;
   S707_WELD_BUFF_DATA81.RBT18_WELD_COUNT := W#16#0;
   S707_WELD_BUFF_DATA81.RBT19_BT_CODE_NO := W#16#0;
   S707_WELD_BUFF_DATA81.RBT19_WELD_COUNT := W#16#0;
   S707_WELD_BUFF_DATA81.RBT20_BT_CODE_NO := W#16#0;
   S707_WELD_BUFF_DATA81.RBT20_WELD_COUNT := W#16#0;
   S707_WELD_BUFF_DATA81.RBT21_BT_CODE_NO := W#16#0;
   S707_WELD_BUFF_DATA81.RBT21_WELD_COUNT := W#16#0;
   S707_WELD_BUFF_DATA81.RBT22_BT_CODE_NO := W#16#0;
   S707_WELD_BUFF_DATA81.RBT22_WELD_COUNT := W#16#0;
   S707_WELD_BUFF_DATA81.RBT23_BT_CODE_NO := W#16#0;
   S707_WELD_BUFF_DATA81.RBT23_WELD_COUNT := W#16#0;
   S707_WELD_BUFF_DATA81.RBT24_BT_CODE_NO := W#16#0;
   S707_WELD_BUFF_DATA81.RBT24_WELD_COUNT := W#16#0;
   S707_WELD_BUFF_DATA81.WELD_DETERMINES_RESULT := W#16#0;
   S707_WELD_BUFF_DATA81.WELD_CHECK_SUM := W#16#0;
   S707_WELD_BUFF_DATA81.SPARE1 := W#16#0;
   S707_WELD_BUFF_DATA91.STATION_MAIN := W#16#0;
   S707_WELD_BUFF_DATA91.DISTINCTION_LH_RH := W#16#0;
   S707_WELD_BUFF_DATA91.STAION_NUMBER := W#16#0;
   S707_WELD_BUFF_DATA91.VIN_NUMBER1 := W#16#0;
   S707_WELD_BUFF_DATA91.VIN_NUMBER2 := W#16#0;
   S707_WELD_BUFF_DATA91.VIN_NUMBER3 := W#16#0;
   S707_WELD_BUFF_DATA91.VIN_NUMBER4 := W#16#0;
   S707_WELD_BUFF_DATA91.SEQ_NUMBER1 := W#16#0;
   S707_WELD_BUFF_DATA91.SEQ_NUMBER2 := W#16#0;
   S707_WELD_BUFF_DATA91.RBT1_BT_CODE_NO := W#16#0;
   S707_WELD_BUFF_DATA91.RBT1_WELD_COUNT := W#16#0;
   S707_WELD_BUFF_DATA91.RBT2_BT_CODE_NO := W#16#0;
   S707_WELD_BUFF_DATA91.RBT2_WELD_COUNT := W#16#0;
   S707_WELD_BUFF_DATA91.RBT3_BT_CODE_NO := W#16#0;
   S707_WELD_BUFF_DATA91.RBT3_WELD_COUNT := W#16#0;
   S707_WELD_BUFF_DATA91.RBT4_BT_CODE_NO := W#16#0;
   S707_WELD_BUFF_DATA91.RBT4_WELD_COUNT := W#16#0;
   S707_WELD_BUFF_DATA91.RBT5_BT_CODE_NO := W#16#0;
   S707_WELD_BUFF_DATA91.RBT5_WELD_COUNT := W#16#0;
   S707_WELD_BUFF_DATA91.RBT6_BT_CODE_NO := W#16#0;
   S707_WELD_BUFF_DATA91.RBT6_WELD_COUNT := W#16#0;
   S707_WELD_BUFF_DATA91.RBT7_BT_CODE_NO := W#16#0;
   S707_WELD_BUFF_DATA91.RBT7_WELD_COUNT := W#16#0;
   S707_WELD_BUFF_DATA91.RBT8_BT_CODE_NO := W#16#0;
   S707_WELD_BUFF_DATA91.RBT8_WELD_COUNT := W#16#0;
   S707_WELD_BUFF_DATA91.RBT9_BT_CODE_NO := W#16#0;
   S707_WELD_BUFF_DATA91.RBT9_WELD_COUNT := W#16#0;
   S707_WELD_BUFF_DATA91.RBT10_BT_CODE_NO := W#16#0;
   S707_WELD_BUFF_DATA91.RBT10_WELD_COUNT := W#16#0;
   S707_WELD_BUFF_DATA91.RBT11_BT_CODE_NO := W#16#0;
   S707_WELD_BUFF_DATA91.RBT11_WELD_COUNT := W#16#0;
   S707_WELD_BUFF_DATA91.RBT12_BT_CODE_NO := W#16#0;
   S707_WELD_BUFF_DATA91.RBT12_WELD_COUNT := W#16#0;
   S707_WELD_BUFF_DATA91.RBT13_BT_CODE_NO := W#16#0;
   S707_WELD_BUFF_DATA91.RBT13_WELD_COUNT := W#16#0;
   S707_WELD_BUFF_DATA91.RBT14_BT_CODE_NO := W#16#0;
   S707_WELD_BUFF_DATA91.RBT14_WELD_COUNT := W#16#0;
   S707_WELD_BUFF_DATA91.RBT15_BT_CODE_NO := W#16#0;
   S707_WELD_BUFF_DATA91.RBT15_WELD_COUNT := W#16#0;
   S707_WELD_BUFF_DATA91.RBT16_BT_CODE_NO := W#16#0;
   S707_WELD_BUFF_DATA91.RBT16_WELD_COUNT := W#16#0;
   S707_WELD_BUFF_DATA91.RBT17_BT_CODE_NO := W#16#0;
   S707_WELD_BUFF_DATA91.RBT17_WELD_COUNT := W#16#0;
   S707_WELD_BUFF_DATA91.RBT18_BT_CODE_NO := W#16#0;
   S707_WELD_BUFF_DATA91.RBT18_WELD_COUNT := W#16#0;
   S707_WELD_BUFF_DATA91.RBT19_BT_CODE_NO := W#16#0;
   S707_WELD_BUFF_DATA91.RBT19_WELD_COUNT := W#16#0;
   S707_WELD_BUFF_DATA91.RBT20_BT_CODE_NO := W#16#0;
   S707_WELD_BUFF_DATA91.RBT20_WELD_COUNT := W#16#0;
   S707_WELD_BUFF_DATA91.RBT21_BT_CODE_NO := W#16#0;
   S707_WELD_BUFF_DATA91.RBT21_WELD_COUNT := W#16#0;
   S707_WELD_BUFF_DATA91.RBT22_BT_CODE_NO := W#16#0;
   S707_WELD_BUFF_DATA91.RBT22_WELD_COUNT := W#16#0;
   S707_WELD_BUFF_DATA91.RBT23_BT_CODE_NO := W#16#0;
   S707_WELD_BUFF_DATA91.RBT23_WELD_COUNT := W#16#0;
   S707_WELD_BUFF_DATA91.RBT24_BT_CODE_NO := W#16#0;
   S707_WELD_BUFF_DATA91.RBT24_WELD_COUNT := W#16#0;
   S707_WELD_BUFF_DATA91.WELD_DETERMINES_RESULT := W#16#0;
   S707_WELD_BUFF_DATA91.WELD_CHECK_SUM := W#16#0;
   S707_WELD_BUFF_DATA91.SPARE1 := W#16#0;
   S707_WELD_BUFF_DATA101.STATION_MAIN := W#16#0;
   S707_WELD_BUFF_DATA101.DISTINCTION_LH_RH := W#16#0;
   S707_WELD_BUFF_DATA101.STAION_NUMBER := W#16#0;
   S707_WELD_BUFF_DATA101.VIN_NUMBER1 := W#16#0;
   S707_WELD_BUFF_DATA101.VIN_NUMBER2 := W#16#0;
   S707_WELD_BUFF_DATA101.VIN_NUMBER3 := W#16#0;
   S707_WELD_BUFF_DATA101.VIN_NUMBER4 := W#16#0;
   S707_WELD_BUFF_DATA101.SEQ_NUMBER1 := W#16#0;
   S707_WELD_BUFF_DATA101.SEQ_NUMBER2 := W#16#0;
   S707_WELD_BUFF_DATA101.RBT1_BT_CODE_NO := W#16#0;
   S707_WELD_BUFF_DATA101.RBT1_WELD_COUNT := W#16#0;
   S707_WELD_BUFF_DATA101.RBT2_BT_CODE_NO := W#16#0;
   S707_WELD_BUFF_DATA101.RBT2_WELD_COUNT := W#16#0;
   S707_WELD_BUFF_DATA101.RBT3_BT_CODE_NO := W#16#0;
   S707_WELD_BUFF_DATA101.RBT3_WELD_COUNT := W#16#0;
   S707_WELD_BUFF_DATA101.RBT4_BT_CODE_NO := W#16#0;
   S707_WELD_BUFF_DATA101.RBT4_WELD_COUNT := W#16#0;
   S707_WELD_BUFF_DATA101.RBT5_BT_CODE_NO := W#16#0;
   S707_WELD_BUFF_DATA101.RBT5_WELD_COUNT := W#16#0;
   S707_WELD_BUFF_DATA101.RBT6_BT_CODE_NO := W#16#0;
   S707_WELD_BUFF_DATA101.RBT6_WELD_COUNT := W#16#0;
   S707_WELD_BUFF_DATA101.RBT7_BT_CODE_NO := W#16#0;
   S707_WELD_BUFF_DATA101.RBT7_WELD_COUNT := W#16#0;
   S707_WELD_BUFF_DATA101.RBT8_BT_CODE_NO := W#16#0;
   S707_WELD_BUFF_DATA101.RBT8_WELD_COUNT := W#16#0;
   S707_WELD_BUFF_DATA101.RBT9_BT_CODE_NO := W#16#0;
   S707_WELD_BUFF_DATA101.RBT9_WELD_COUNT := W#16#0;
   S707_WELD_BUFF_DATA101.RBT10_BT_CODE_NO := W#16#0;
   S707_WELD_BUFF_DATA101.RBT10_WELD_COUNT := W#16#0;
   S707_WELD_BUFF_DATA101.RBT11_BT_CODE_NO := W#16#0;
   S707_WELD_BUFF_DATA101.RBT11_WELD_COUNT := W#16#0;
   S707_WELD_BUFF_DATA101.RBT12_BT_CODE_NO := W#16#0;
   S707_WELD_BUFF_DATA101.RBT12_WELD_COUNT := W#16#0;
   S707_WELD_BUFF_DATA101.RBT13_BT_CODE_NO := W#16#0;
   S707_WELD_BUFF_DATA101.RBT13_WELD_COUNT := W#16#0;
   S707_WELD_BUFF_DATA101.RBT14_BT_CODE_NO := W#16#0;
   S707_WELD_BUFF_DATA101.RBT14_WELD_COUNT := W#16#0;
   S707_WELD_BUFF_DATA101.RBT15_BT_CODE_NO := W#16#0;
   S707_WELD_BUFF_DATA101.RBT15_WELD_COUNT := W#16#0;
   S707_WELD_BUFF_DATA101.RBT16_BT_CODE_NO := W#16#0;
   S707_WELD_BUFF_DATA101.RBT16_WELD_COUNT := W#16#0;
   S707_WELD_BUFF_DATA101.RBT17_BT_CODE_NO := W#16#0;
   S707_WELD_BUFF_DATA101.RBT17_WELD_COUNT := W#16#0;
   S707_WELD_BUFF_DATA101.RBT18_BT_CODE_NO := W#16#0;
   S707_WELD_BUFF_DATA101.RBT18_WELD_COUNT := W#16#0;
   S707_WELD_BUFF_DATA101.RBT19_BT_CODE_NO := W#16#0;
   S707_WELD_BUFF_DATA101.RBT19_WELD_COUNT := W#16#0;
   S707_WELD_BUFF_DATA101.RBT20_BT_CODE_NO := W#16#0;
   S707_WELD_BUFF_DATA101.RBT20_WELD_COUNT := W#16#0;
   S707_WELD_BUFF_DATA101.RBT21_BT_CODE_NO := W#16#0;
   S707_WELD_BUFF_DATA101.RBT21_WELD_COUNT := W#16#0;
   S707_WELD_BUFF_DATA101.RBT22_BT_CODE_NO := W#16#0;
   S707_WELD_BUFF_DATA101.RBT22_WELD_COUNT := W#16#0;
   S707_WELD_BUFF_DATA101.RBT23_BT_CODE_NO := W#16#0;
   S707_WELD_BUFF_DATA101.RBT23_WELD_COUNT := W#16#0;
   S707_WELD_BUFF_DATA101.RBT24_BT_CODE_NO := W#16#0;
   S707_WELD_BUFF_DATA101.RBT24_WELD_COUNT := W#16#0;
   S707_WELD_BUFF_DATA101.WELD_DETERMINES_RESULT := W#16#0;
   S707_WELD_BUFF_DATA101.WELD_CHECK_SUM := W#16#0;
   S707_WELD_BUFF_DATA101.SPARE1 := W#16#0;
END_DATA_BLOCK

DATA_BLOCK DB 45
TITLE =
VERSION : 0.1


  STRUCT
   STAT0 : ARRAY  [0 .. 99 ] OF WORD  := W#16#0;
   STAT01 : ARRAY  [0 .. 99 ] OF WORD  := W#16#0;
   STAT02 : ARRAY  [0 .. 99 ] OF WORD  := W#16#0;
  END_STRUCT ;
BEGIN
   STAT0[0] := W#16#0;
   STAT0[1] := W#16#0;
   STAT0[2] := W#16#0;
   STAT0[3] := W#16#0;
   STAT0[4] := W#16#0;
   STAT0[5] := W#16#0;
   STAT0[6] := W#16#0;
   STAT0[7] := W#16#0;
   STAT0[8] := W#16#0;
   STAT0[9] := W#16#0;
   STAT0[10] := W#16#0;
   STAT0[11] := W#16#0;
   STAT0[12] := W#16#0;
   STAT0[13] := W#16#0;
   STAT0[14] := W#16#0;
   STAT0[15] := W#16#0;
   STAT0[16] := W#16#0;
   STAT0[17] := W#16#0;
   STAT0[18] := W#16#0;
   STAT0[19] := W#16#0;
   STAT0[20] := W#16#0;
   STAT0[21] := W#16#0;
   STAT0[22] := W#16#0;
   STAT0[23] := W#16#0;
   STAT0[24] := W#16#0;
   STAT0[25] := W#16#0;
   STAT0[26] := W#16#0;
   STAT0[27] := W#16#0;
   STAT0[28] := W#16#0;
   STAT0[29] := W#16#0;
   STAT0[30] := W#16#0;
   STAT0[31] := W#16#0;
   STAT0[32] := W#16#0;
   STAT0[33] := W#16#0;
   STAT0[34] := W#16#0;
   STAT0[35] := W#16#0;
   STAT0[36] := W#16#0;
   STAT0[37] := W#16#0;
   STAT0[38] := W#16#0;
   STAT0[39] := W#16#0;
   STAT0[40] := W#16#0;
   STAT0[41] := W#16#0;
   STAT0[42] := W#16#0;
   STAT0[43] := W#16#0;
   STAT0[44] := W#16#0;
   STAT0[45] := W#16#0;
   STAT0[46] := W#16#0;
   STAT0[47] := W#16#0;
   STAT0[48] := W#16#0;
   STAT0[49] := W#16#0;
   STAT0[50] := W#16#0;
   STAT0[51] := W#16#0;
   STAT0[52] := W#16#0;
   STAT0[53] := W#16#0;
   STAT0[54] := W#16#0;
   STAT0[55] := W#16#0;
   STAT0[56] := W#16#0;
   STAT0[57] := W#16#0;
   STAT0[58] := W#16#0;
   STAT0[59] := W#16#0;
   STAT0[60] := W#16#0;
   STAT0[61] := W#16#0;
   STAT0[62] := W#16#0;
   STAT0[63] := W#16#0;
   STAT0[64] := W#16#0;
   STAT0[65] := W#16#0;
   STAT0[66] := W#16#0;
   STAT0[67] := W#16#0;
   STAT0[68] := W#16#0;
   STAT0[69] := W#16#0;
   STAT0[70] := W#16#0;
   STAT0[71] := W#16#0;
   STAT0[72] := W#16#0;
   STAT0[73] := W#16#0;
   STAT0[74] := W#16#0;
   STAT0[75] := W#16#0;
   STAT0[76] := W#16#0;
   STAT0[77] := W#16#0;
   STAT0[78] := W#16#0;
   STAT0[79] := W#16#0;
   STAT0[80] := W#16#0;
   STAT0[81] := W#16#0;
   STAT0[82] := W#16#0;
   STAT0[83] := W#16#0;
   STAT0[84] := W#16#0;
   STAT0[85] := W#16#0;
   STAT0[86] := W#16#0;
   STAT0[87] := W#16#0;
   STAT0[88] := W#16#0;
   STAT0[89] := W#16#0;
   STAT0[90] := W#16#0;
   STAT0[91] := W#16#0;
   STAT0[92] := W#16#0;
   STAT0[93] := W#16#0;
   STAT0[94] := W#16#0;
   STAT0[95] := W#16#0;
   STAT0[96] := W#16#0;
   STAT0[97] := W#16#0;
   STAT0[98] := W#16#0;
   STAT0[99] := W#16#0;
   STAT01[0] := W#16#0;
   STAT01[1] := W#16#0;
   STAT01[2] := W#16#0;
   STAT01[3] := W#16#0;
   STAT01[4] := W#16#0;
   STAT01[5] := W#16#0;
   STAT01[6] := W#16#0;
   STAT01[7] := W#16#0;
   STAT01[8] := W#16#0;
   STAT01[9] := W#16#0;
   STAT01[10] := W#16#14;
   STAT01[11] := W#16#1803;
   STAT01[12] := W#16#210A;
   STAT01[13] := W#16#8010;
   STAT01[14] := W#16#1654;
   STAT01[15] := W#16#0;
   STAT01[16] := W#16#0;
   STAT01[17] := W#16#0;
   STAT01[18] := W#16#0;
   STAT01[19] := W#16#0;
   STAT01[20] := W#16#14;
   STAT01[21] := W#16#1802;
   STAT01[22] := W#16#2122;
   STAT01[23] := W#16#8002;
   STAT01[24] := W#16#2654;
   STAT01[25] := W#16#8001;
   STAT01[26] := W#16#0;
   STAT01[27] := W#16#0;
   STAT01[28] := W#16#0;
   STAT01[29] := W#16#0;
   STAT01[30] := W#16#14;
   STAT01[31] := W#16#1801;
   STAT01[32] := W#16#2122;
   STAT01[33] := W#16#8004;
   STAT01[34] := W#16#1654;
   STAT01[35] := W#16#0;
   STAT01[36] := W#16#0;
   STAT01[37] := W#16#0;
   STAT01[38] := W#16#0;
   STAT01[39] := W#16#0;
   STAT01[40] := W#16#14;
   STAT01[41] := W#16#1800;
   STAT01[42] := W#16#210A;
   STAT01[43] := W#16#8008;
   STAT01[44] := W#16#1654;
   STAT01[45] := W#16#0;
   STAT01[46] := W#16#0;
   STAT01[47] := W#16#0;
   STAT01[48] := W#16#0;
   STAT01[49] := W#16#0;
   STAT01[50] := W#16#14;
   STAT01[51] := W#16#1799;
   STAT01[52] := W#16#2114;
   STAT01[53] := W#16#8004;
   STAT01[54] := W#16#5254;
   STAT01[55] := W#16#1;
   STAT01[56] := W#16#0;
   STAT01[57] := W#16#0;
   STAT01[58] := W#16#0;
   STAT01[59] := W#16#0;
   STAT01[60] := W#16#14;
   STAT01[61] := W#16#1798;
   STAT01[62] := W#16#2122;
   STAT01[63] := W#16#8004;
   STAT01[64] := W#16#1654;
   STAT01[65] := W#16#0;
   STAT01[66] := W#16#0;
   STAT01[67] := W#16#0;
   STAT01[68] := W#16#0;
   STAT01[69] := W#16#0;
   STAT01[70] := W#16#14;
   STAT01[71] := W#16#1797;
   STAT01[72] := W#16#210A;
   STAT01[73] := W#16#8008;
   STAT01[74] := W#16#1616;
   STAT01[75] := W#16#0;
   STAT01[76] := W#16#0;
   STAT01[77] := W#16#0;
   STAT01[78] := W#16#0;
   STAT01[79] := W#16#0;
   STAT01[80] := W#16#14;
   STAT01[81] := W#16#1796;
   STAT01[82] := W#16#210A;
   STAT01[83] := W#16#8010;
   STAT01[84] := W#16#1654;
   STAT01[85] := W#16#0;
   STAT01[86] := W#16#0;
   STAT01[87] := W#16#0;
   STAT01[88] := W#16#0;
   STAT01[89] := W#16#0;
   STAT01[90] := W#16#14;
   STAT01[91] := W#16#1795;
   STAT01[92] := W#16#2122;
   STAT01[93] := W#16#8002;
   STAT01[94] := W#16#6254;
   STAT01[95] := W#16#8001;
   STAT01[96] := W#16#0;
   STAT01[97] := W#16#0;
   STAT01[98] := W#16#0;
   STAT01[99] := W#16#0;
   STAT02[0] := W#16#0;
   STAT02[1] := W#16#0;
   STAT02[2] := W#16#0;
   STAT02[3] := W#16#0;
   STAT02[4] := W#16#0;
   STAT02[5] := W#16#0;
   STAT02[6] := W#16#0;
   STAT02[7] := W#16#0;
   STAT02[8] := W#16#0;
   STAT02[9] := W#16#0;
   STAT02[10] := W#16#14;
   STAT02[11] := W#16#1802;
   STAT02[12] := W#16#2122;
   STAT02[13] := W#16#8002;
   STAT02[14] := W#16#2654;
   STAT02[15] := W#16#8001;
   STAT02[16] := W#16#0;
   STAT02[17] := W#16#0;
   STAT02[18] := W#16#0;
   STAT02[19] := W#16#0;
   STAT02[20] := W#16#14;
   STAT02[21] := W#16#1801;
   STAT02[22] := W#16#2122;
   STAT02[23] := W#16#8004;
   STAT02[24] := W#16#1654;
   STAT02[25] := W#16#0;
   STAT02[26] := W#16#0;
   STAT02[27] := W#16#0;
   STAT02[28] := W#16#0;
   STAT02[29] := W#16#0;
   STAT02[30] := W#16#14;
   STAT02[31] := W#16#1800;
   STAT02[32] := W#16#210A;
   STAT02[33] := W#16#8008;
   STAT02[34] := W#16#1654;
   STAT02[35] := W#16#0;
   STAT02[36] := W#16#0;
   STAT02[37] := W#16#0;
   STAT02[38] := W#16#0;
   STAT02[39] := W#16#0;
   STAT02[40] := W#16#14;
   STAT02[41] := W#16#1799;
   STAT02[42] := W#16#2114;
   STAT02[43] := W#16#8004;
   STAT02[44] := W#16#5254;
   STAT02[45] := W#16#1;
   STAT02[46] := W#16#0;
   STAT02[47] := W#16#0;
   STAT02[48] := W#16#0;
   STAT02[49] := W#16#0;
   STAT02[50] := W#16#14;
   STAT02[51] := W#16#1798;
   STAT02[52] := W#16#2122;
   STAT02[53] := W#16#8004;
   STAT02[54] := W#16#1654;
   STAT02[55] := W#16#0;
   STAT02[56] := W#16#0;
   STAT02[57] := W#16#0;
   STAT02[58] := W#16#0;
   STAT02[59] := W#16#0;
   STAT02[60] := W#16#14;
   STAT02[61] := W#16#1797;
   STAT02[62] := W#16#210A;
   STAT02[63] := W#16#8008;
   STAT02[64] := W#16#1616;
   STAT02[65] := W#16#0;
   STAT02[66] := W#16#0;
   STAT02[67] := W#16#0;
   STAT02[68] := W#16#0;
   STAT02[69] := W#16#0;
   STAT02[70] := W#16#14;
   STAT02[71] := W#16#1796;
   STAT02[72] := W#16#210A;
   STAT02[73] := W#16#8010;
   STAT02[74] := W#16#1654;
   STAT02[75] := W#16#0;
   STAT02[76] := W#16#0;
   STAT02[77] := W#16#0;
   STAT02[78] := W#16#0;
   STAT02[79] := W#16#0;
   STAT02[80] := W#16#14;
   STAT02[81] := W#16#1795;
   STAT02[82] := W#16#2122;
   STAT02[83] := W#16#8002;
   STAT02[84] := W#16#6254;
   STAT02[85] := W#16#8001;
   STAT02[86] := W#16#0;
   STAT02[87] := W#16#0;
   STAT02[88] := W#16#0;
   STAT02[89] := W#16#0;
   STAT02[90] := W#16#14;
   STAT02[91] := W#16#1794;
   STAT02[92] := W#16#2122;
   STAT02[93] := W#16#8004;
   STAT02[94] := W#16#1654;
   STAT02[95] := W#16#0;
   STAT02[96] := W#16#0;
   STAT02[97] := W#16#0;
   STAT02[98] := W#16#0;
   STAT02[99] := W#16#0;
END_DATA_BLOCK

DATA_BLOCK DB 51
TITLE =
VERSION : 0.1


  STRUCT
   S_705 : STRUCT
    M_AUTO_SEL : BOOL ;
    M_MANUAL_SEL : BOOL ;
    M_READY_PB : BOOL ;
    M_AUTO_RUN_PB : BOOL ;
    M_WORK_COMP_SET_PB : BOOL ;
    M_WORK_COMP_RST_PB : BOOL ;
    M_HOME_POS_PB : BOOL ;
    M_TIP_DRESS_PB : BOOL ;
    HOOK_PIN_SEL : BOOL ;
    DAECHA_LOCK_SEL : BOOL ;
    ELE_SEL : BOOL ;
    AIR_ELE_SEL : BOOL ;
    SPARE13 : BOOL ;
    SPARE14 : BOOL ;
    SPARE15 : BOOL ;
    SPARE16 : BOOL ;
    SPARE17 : BOOL ;
    SPARE18 : BOOL ;
    SPARE19 : BOOL ;
    SPARE20 : BOOL ;
    SPARE21 : BOOL ;
    SPARE22 : BOOL ;
    SPARE23 : BOOL ;
    SPARE24 : BOOL ;
    SPARE25 : BOOL ;
    SPARE26 : BOOL ;
    SPARE27 : BOOL ;
    SPARE28 : BOOL ;
    SPARE29 : BOOL ;
    SPARE30 : BOOL ;
    M_ADV_PB : BOOL ;
    M_RET_PB : BOOL ;
    LM_DC_PIN_SEL : BOOL ;
    LM_DC_1ST_CLAMP1_SEL : BOOL ;
    LM_DC_1ST_CLAMP2_SEL : BOOL ;
    LM_DC_1ST_CLAMP3_SEL : BOOL ;
    LM_DC_1ST_CLAMP4_SEL : BOOL ;
    LM_DC_2ND_CLAMP1_SEL : BOOL ;
    LM_DC_2ND_CLAMP2_SEL : BOOL ;
    LM_DC_2ND_CLAMP3_SEL : BOOL ;
    LM_DC_2ND_CLAMP4_SEL : BOOL ;
    LM_DC_2ND_CLAMP5_SEL : BOOL ;
    LM_DC_DR_STK_PIN_SEL : BOOL ;
    LM_DC_OTR_CLAMP_SEL : BOOL ;
    LM_DC_ASSY_CLAMP_SEL : BOOL ;
    LM_DC_FF_PIN_SEL : BOOL ;
    LM_DC_FF_CLAMP_SEL : BOOL ;
    LM_DC_2ND_CLAMP6_SEL : BOOL ;
    SPARE50 : BOOL ;
    SPARE51 : BOOL ;
    SPARE52 : BOOL ;
    SPARE53 : BOOL ;
    SPARE54 : BOOL ;
    SPARE55 : BOOL ;
    SPARE56 : BOOL ;
    SPARE57 : BOOL ;
    SPARE58 : BOOL ;
    SPARE59 : BOOL ;
    SPARE60 : BOOL ;
    SPARE61 : BOOL ;
    SPARE62 : BOOL ;
    SPARE63 : BOOL ;
    LM_DC_M_ADV_PB : BOOL ;
    LM_DC_M_RET_PB : BOOL ;
    TL_DC_PIN_SEL : BOOL ;
    TL_DC_LATCH1_SEL : BOOL ;
    TL_DC_1ST_CLAMP_SEL : BOOL ;
    TL_DC_2ND_CLAMP_SEL : BOOL ;
    TL_DC_U261_SEL : BOOL ;
    TL_DC_U261_CLAMP_SEL : BOOL ;
    TL_DC_U269_UP_DN_SEL : BOOL ;
    TL_DC_U269_CLAMP_SEL : BOOL ;
    TL_DC_3RD_CLAMP_SEL : BOOL ;
    TL_DC_U262_1_UP_DN_SEL : BOOL ;
    TL_DC_U262_1_SEL : BOOL ;
    TL_DC_U262_1_CLAMP_SEL : BOOL ;
    TL_DC_U261_2_CLAMP_SEL : BOOL ;
    SPARE79 : BOOL ;
    SPARE80 : BOOL ;
    SPARE81 : BOOL ;
    SPARE82 : BOOL ;
    SPARE83 : BOOL ;
    SPARE84 : BOOL ;
    SPARE85 : BOOL ;
    SPARE86 : BOOL ;
    SPARE87 : BOOL ;
    SPARE88 : BOOL ;
    SPARE89 : BOOL ;
    SPARE90 : BOOL ;
    SPARE91 : BOOL ;
    SPARE92 : BOOL ;
    SPARE93 : BOOL ;
    SPARE94 : BOOL ;
    SPARE95 : BOOL ;
    TL_DC_M_ADV_PB : BOOL ;
    TL_DC_M_RET_PB : BOOL ;
    SPARE98 : BOOL ;
    SPARE99 : BOOL ;
    SPARE100 : BOOL ;
    SPARE101 : BOOL ;
    SPARE102 : BOOL ;
    SPARE103 : BOOL ;
    SPARE104 : BOOL ;
    SPARE105 : BOOL ;
    SPARE106 : BOOL ;
    SPARE107 : BOOL ;
    SPARE108 : BOOL ;
    SPARE109 : BOOL ;
    SPARE110 : BOOL ;
    SPARE111 : BOOL ;
    SPARE112 : BOOL ;
    SPARE113 : BOOL ;
    SPARE114 : BOOL ;
    SPARE115 : BOOL ;
    SPARE116 : BOOL ;
    SPARE117 : BOOL ;
    SPARE118 : BOOL ;
    SPARE119 : BOOL ;
    SPARE120 : BOOL ;
    SPARE121 : BOOL ;
    SPARE122 : BOOL ;
    SPARE123 : BOOL ;
    SPARE124 : BOOL ;
    SPARE125 : BOOL ;
    SPARE126 : BOOL ;
    SPARE127 : BOOL ;
    SPARE128 : BOOL ;
    SPARE129 : BOOL ;
    SPARE130 : BOOL ;
    SPARE131 : BOOL ;
    SPARE132 : BOOL ;
    SPARE133 : BOOL ;
    SPARE134 : BOOL ;
    SPARE135 : BOOL ;
    SPARE136 : BOOL ;
    SPARE137 : BOOL ;
    SPARE138 : BOOL ;
    SPARE139 : BOOL ;
    SPARE140 : BOOL ;
    SPARE141 : BOOL ;
    SPARE142 : BOOL ;
    SPARE143 : BOOL ;
    SPARE144 : BOOL ;
    SPARE145 : BOOL ;
    SPARE146 : BOOL ;
    SPARE147 : BOOL ;
    SPARE148 : BOOL ;
    SPARE149 : BOOL ;
    SPARE150 : BOOL ;
    SPARE151 : BOOL ;
    SPARE152 : BOOL ;
    SPARE153 : BOOL ;
    SPARE154 : BOOL ;
    SPARE155 : BOOL ;
    SPARE156 : BOOL ;
    SPARE157 : BOOL ;
    SPARE158 : BOOL ;
    SPARE159 : BOOL ;
    SPARE160 : BOOL ;
    S705_R2_R3_WORK_COMP_SET : BOOL ;
    HOOK_PIN_UP_LP : WORD ;
    HOOK_PIN_DOWN_LP : WORD ;
    DAECHA_LOCK_ADV_LP : WORD ;
    DAECHA_LOCK_RET_LP : WORD ;
    ELE_ADV_LP : WORD ;
    ELE_RET_LP : WORD ;
    AIR_ELE_ADV_LP : WORD ;
    AIR_ELE_RET_LP : WORD ;
    SP_WORD19 : WORD ;
    SP_WORD20 : WORD ;
    LM_DC_PIN_UP_LP : WORD ;
    LM_DC_PIN_DOWN_LP : WORD ;
    LM_DC_1ST_CLAMP1_ADV_LP : WORD ;
    LM_DC_1ST_CLAMP1_RET_LP : WORD ;
    LM_DC_1ST_CLAMP2_ADV_LP : WORD ;
    LM_DC_1ST_CLAMP2_RET_LP : WORD ;
    LM_DC_1ST_CLAMP3_ADV_LP : WORD ;
    LM_DC_1ST_CLAMP3_RET_LP : WORD ;
    LM_DC_1ST_CLAMP4_ADV_LP : WORD ;
    LM_DC_1ST_CLAMP4_RET_LP : WORD ;
    LM_DC_2ND_CLAMP1_ADV_LP : WORD ;
    LM_DC_2ND_CLAMP1_RET_LP : WORD ;
    LM_DC_2ND_CLAMP2_ADV_LP : WORD ;
    LM_DC_2ND_CLAMP2_RET_LP : WORD ;
    LM_DC_2ND_CLAMP3_ADV_LP : WORD ;
    LM_DC_2ND_CLAMP3_RET_LP : WORD ;
    LM_DC_2ND_CLAMP4_ADV_LP : WORD ;
    LM_DC_2ND_CLAMP4_RET_LP : WORD ;
    LM_DC_2ND_CLAMP5_ADV_LP : WORD ;
    LM_DC_2ND_CLAMP5_RET_LP : WORD ;
    LM_DC_DR_STK_PIN_UP_LP : WORD ;
    LM_DC_DR_STK_PIN_DOWN_LP : WORD ;
    LM_DC_OTR_CLAMP_ADV_LP : WORD ;
    LM_DC_OTR_CLAMP_RET_LP : WORD ;
    LM_DC_ASSY_CLAMP_ADV_LP : WORD ;
    LM_DC_ASSY_CLAMP_RET_LP : WORD ;
    LM_DC_FF_PIN_UP_LP : WORD ;
    LM_DC_FF_PIN_DOWN_LP : WORD ;
    LM_DC_FF_CLAMP_ADV_LP : WORD ;
    LM_DC_FF_CLAMP_RET_LP : WORD ;
    LM_DC_2ND_CLAMP6_ADV_LP : WORD ;
    LM_DC_2ND_CLAMP6_RET_LP : WORD ;
    LM_DC_2ND_CLAMP7_ADV_LP : WORD ;
    LM_DC_2ND_CLAMP7_RET_LP : WORD ;
    LM_DC_1ST_CLAMP5_ADV_LP : WORD ;
    LM_DC_1ST_CLAMP5_RET_LP : WORD ;
    SP_WORD68 : WORD ;
    SP_WORD69 : WORD ;
    SP_WORD70 : WORD ;
    SP_WORD71 : WORD ;
    TL_DC_PIN_UP_LP : WORD ;
    TL_DC_PIN_DOWN_LP : WORD ;
    TL_DC_LATCH1_ADV_LP : WORD ;
    TL_DC_LATCH1_RET_LP : WORD ;
    TL_DC_LATCH2_ADV_LP : WORD ;
    TL_DC_LATCH2_RET_LP : WORD ;
    TL_DC_1ST_CLAMP1_ADV_LP : WORD ;
    TL_DC_1ST_CLAMP1_RET_LP : WORD ;
    TL_DC_1ST_CLAMP2_ADV_LP : WORD ;
    TL_DC_1ST_CLAMP2_RET_LP : WORD ;
    TL_DC_1ST_CLAMP3_ADV_LP : WORD ;
    TL_DC_1ST_CLAMP3_RET_LP : WORD ;
    TL_DC_2ND_CLAMP1_ADV_LP : WORD ;
    TL_DC_2ND_CLAMP1_RET_LP : WORD ;
    TL_DC_2ND_CLAMP2_ADV_LP : WORD ;
    TL_DC_2ND_CLAMP2_RET_LP : WORD ;
    TL_DC_U261_ADV_LP : WORD ;
    TL_DC_U261_RET_LP : WORD ;
    TL_DC_U261_CLAMP_ADV_LP : WORD ;
    TL_DC_U261_CLAMP_RET_LP : WORD ;
    TL_DC_U269_UP_LP : WORD ;
    TL_DC_U269_DOWN_LP : WORD ;
    TL_DC_U269_CLAMP_ADV_LP : WORD ;
    TL_DC_U269_CLAMP_RET_LP : WORD ;
    TL_DC_3RD_CLAMP_ADV_LP : WORD ;
    TL_DC_3RD_CLAMP_RET_LP : WORD ;
    TL_DC_U262_1_UP_LP : WORD ;
    TL_DC_U262_1_DOWN_LP : WORD ;
    TL_DC_U262_1_ADV_LP : WORD ;
    TL_DC_U262_1_RET_LP : WORD ;
    TL_DC_U262_1_CLP_ADV_LP : WORD ;
    TL_DC_U262_1_CLP_RET_LP : WORD ;
    TL_DC_U261_2_CLP_ADV_LP : WORD ;
    TL_DC_U261_2_CLP_RET_LP : WORD ;
    SP_WORD106 : WORD ;
    SP_WORD107 : WORD ;
    SP_WORD108 : WORD ;
    SP_WORD109 : WORD ;
    SP_WORD110 : WORD ;
    SP_WORD111 : WORD ;
   END_STRUCT ;
   S_706 : STRUCT
    M_AUTO_SEL : BOOL ;
    M_MANUAL_SEL : BOOL ;
    M_READY_PB : BOOL ;
    M_AUTO_RUN_PB : BOOL ;
    M_WORK_COMP_SET_PB : BOOL ;
    M_WORK_COMP_RST_PB : BOOL ;
    M_HOME_POS_PB : BOOL ;
    M_TIP_DRESS_PB : BOOL ;
    HOOK_PIN_SEL : BOOL ;
    DAECHA_LOCK_SEL : BOOL ;
    ELE_SEL : BOOL ;
    AIR_ELE_SEL : BOOL ;
    SPARE13 : BOOL ;
    SPARE14 : BOOL ;
    SPARE15 : BOOL ;
    SPARE16 : BOOL ;
    SPARE17 : BOOL ;
    SPARE18 : BOOL ;
    SPARE19 : BOOL ;
    SPARE20 : BOOL ;
    SPARE21 : BOOL ;
    SPARE22 : BOOL ;
    SPARE23 : BOOL ;
    SPARE24 : BOOL ;
    SPARE25 : BOOL ;
    SPARE26 : BOOL ;
    SPARE27 : BOOL ;
    SPARE28 : BOOL ;
    SPARE29 : BOOL ;
    SPARE30 : BOOL ;
    M_ADV_PB : BOOL ;
    M_RET_PB : BOOL ;
    LM_DC_PIN_SEL : BOOL ;
    LM_DC_1ST_CLAMP1_SEL : BOOL ;
    LM_DC_1ST_CLAMP2_SEL : BOOL ;
    LM_DC_1ST_CLAMP3_SEL : BOOL ;
    LM_DC_1ST_CLAMP4_SEL : BOOL ;
    LM_DC_2ND_CLAMP1_SEL : BOOL ;
    LM_DC_2ND_CLAMP2_SEL : BOOL ;
    LM_DC_2ND_CLAMP3_SEL : BOOL ;
    LM_DC_2ND_CLAMP4_SEL : BOOL ;
    LM_DC_2ND_CLAMP5_SEL : BOOL ;
    LM_DC_DR_STK_PIN_SEL : BOOL ;
    LM_DC_OTR_CLAMP_SEL : BOOL ;
    LM_DC_ASSY_CLAMP_SEL : BOOL ;
    LM_DC_FF_PIN_SEL : BOOL ;
    LM_DC_FF_CLAMP_SEL : BOOL ;
    LM_DC_2ND_CLAMP6_SEL : BOOL ;
    SPARE50 : BOOL ;
    SPARE51 : BOOL ;
    SPARE52 : BOOL ;
    SPARE53 : BOOL ;
    SPARE54 : BOOL ;
    SPARE55 : BOOL ;
    SPARE56 : BOOL ;
    SPARE57 : BOOL ;
    SPARE58 : BOOL ;
    SPARE59 : BOOL ;
    SPARE60 : BOOL ;
    SPARE61 : BOOL ;
    SPARE62 : BOOL ;
    SPARE63 : BOOL ;
    LM_DC_M_ADV_PB : BOOL ;
    LM_DC_M_RET_PB : BOOL ;
    TL_DC_PIN_SEL : BOOL ;
    TL_DC_LATCH1_SEL : BOOL ;
    TL_DC_1ST_CLAMP_SEL : BOOL ;
    TL_DC_2ND_CLAMP_SEL : BOOL ;
    TL_DC_U261_SEL : BOOL ;
    TL_DC_U261_CLAMP_SEL : BOOL ;
    TL_DC_U269_UP_DN_SEL : BOOL ;
    TL_DC_U269_CLAMP_SEL : BOOL ;
    TL_DC_3RD_CLAMP_SEL : BOOL ;
    TL_DC_U262_1_UP_DN_SEL : BOOL ;
    TL_DC_U262_1_SEL : BOOL ;
    TL_DC_U262_1_CLAMP_SEL : BOOL ;
    TL_DC_U261_2_CLAMP_SEL : BOOL ;
    SPARE79 : BOOL ;
    SPARE80 : BOOL ;
    SPARE81 : BOOL ;
    SPARE82 : BOOL ;
    SPARE83 : BOOL ;
    SPARE84 : BOOL ;
    SPARE85 : BOOL ;
    SPARE86 : BOOL ;
    SPARE87 : BOOL ;
    SPARE88 : BOOL ;
    SPARE89 : BOOL ;
    SPARE90 : BOOL ;
    SPARE91 : BOOL ;
    SPARE92 : BOOL ;
    SPARE93 : BOOL ;
    SPARE94 : BOOL ;
    SPARE95 : BOOL ;
    TL_DC_M_ADV_PB : BOOL ;
    TL_DC_M_RET_PB : BOOL ;
    SPARE98 : BOOL ;
    SPARE99 : BOOL ;
    SPARE100 : BOOL ;
    SPARE101 : BOOL ;
    SPARE102 : BOOL ;
    SPARE103 : BOOL ;
    SPARE104 : BOOL ;
    SPARE105 : BOOL ;
    SPARE106 : BOOL ;
    SPARE107 : BOOL ;
    SPARE108 : BOOL ;
    SPARE109 : BOOL ;
    SPARE110 : BOOL ;
    SPARE111 : BOOL ;
    SPARE112 : BOOL ;
    SPARE113 : BOOL ;
    SPARE114 : BOOL ;
    SPARE115 : BOOL ;
    SPARE116 : BOOL ;
    SPARE117 : BOOL ;
    SPARE118 : BOOL ;
    SPARE119 : BOOL ;
    SPARE120 : BOOL ;
    SPARE121 : BOOL ;
    SPARE122 : BOOL ;
    SPARE123 : BOOL ;
    SPARE124 : BOOL ;
    SPARE125 : BOOL ;
    SPARE126 : BOOL ;
    SPARE127 : BOOL ;
    SPARE128 : BOOL ;
    SPARE129 : BOOL ;
    SPARE130 : BOOL ;
    SPARE131 : BOOL ;
    SPARE132 : BOOL ;
    SPARE133 : BOOL ;
    SPARE134 : BOOL ;
    SPARE135 : BOOL ;
    SPARE136 : BOOL ;
    SPARE137 : BOOL ;
    SPARE138 : BOOL ;
    SPARE139 : BOOL ;
    SPARE140 : BOOL ;
    SPARE141 : BOOL ;
    SPARE142 : BOOL ;
    SPARE143 : BOOL ;
    SPARE144 : BOOL ;
    SPARE145 : BOOL ;
    SPARE146 : BOOL ;
    SPARE147 : BOOL ;
    SPARE148 : BOOL ;
    SPARE149 : BOOL ;
    SPARE150 : BOOL ;
    SPARE151 : BOOL ;
    SPARE152 : BOOL ;
    SPARE153 : BOOL ;
    SPARE154 : BOOL ;
    SPARE155 : BOOL ;
    SPARE156 : BOOL ;
    SPARE157 : BOOL ;
    SPARE158 : BOOL ;
    SPARE159 : BOOL ;
    SPARE160 : BOOL ;
    SPARE161 : BOOL ;
    HOOK_PIN_UP_LP : WORD ;
    HOOK_PIN_DOWN_LP : WORD ;
    DAECHA_LOCK_ADV_LP : WORD ;
    DAECHA_LOCK_RET_LP : WORD ;
    ELE_ADV_LP : WORD ;
    ELE_RET_LP : WORD ;
    AIR_ELE_ADV_LP : WORD ;
    AIR_ELE_RET_LP : WORD ;
    SP_WORD19 : WORD ;
    SP_WORD20 : WORD ;
    LM_DC_PIN_UP_LP : WORD ;
    LM_DC_PIN_DOWN_LP : WORD ;
    LM_DC_1ST_CLAMP1_ADV_LP : WORD ;
    LM_DC_1ST_CLAMP1_RET_LP : WORD ;
    LM_DC_1ST_CLAMP2_ADV_LP : WORD ;
    LM_DC_1ST_CLAMP2_RET_LP : WORD ;
    LM_DC_1ST_CLAMP3_ADV_LP : WORD ;
    LM_DC_1ST_CLAMP3_RET_LP : WORD ;
    LM_DC_1ST_CLAMP4_ADV_LP : WORD ;
    LM_DC_1ST_CLAMP4_RET_LP : WORD ;
    LM_DC_2ND_CLAMP1_ADV_LP : WORD ;
    LM_DC_2ND_CLAMP1_RET_LP : WORD ;
    LM_DC_2ND_CLAMP2_ADV_LP : WORD ;
    LM_DC_2ND_CLAMP2_RET_LP : WORD ;
    LM_DC_2ND_CLAMP3_ADV_LP : WORD ;
    LM_DC_2ND_CLAMP3_RET_LP : WORD ;
    LM_DC_2ND_CLAMP4_ADV_LP : WORD ;
    LM_DC_2ND_CLAMP4_RET_LP : WORD ;
    LM_DC_2ND_CLAMP5_ADV_LP : WORD ;
    LM_DC_2ND_CLAMP5_RET_LP : WORD ;
    LM_DC_DR_STK_PIN_UP_LP : WORD ;
    LM_DC_DR_STK_PIN_DOWN_LP : WORD ;
    LM_DC_OTR_CLAMP_ADV_LP : WORD ;
    LM_DC_OTR_CLAMP_RET_LP : WORD ;
    LM_DC_ASSY_CLAMP_ADV_LP : WORD ;
    LM_DC_ASSY_CLAMP_RET_LP : WORD ;
    LM_DC_FF_PIN_UP_LP : WORD ;
    LM_DC_FF_PIN_DOWN_LP : WORD ;
    LM_DC_FF_CLAMP_ADV_LP : WORD ;
    LM_DC_FF_CLAMP_RET_LP : WORD ;
    LM_DC_2ND_CLAMP6_ADV_LP : WORD ;
    LM_DC_2ND_CLAMP6_RET_LP : WORD ;
    LM_DC_2ND_CLAMP7_ADV_LP : WORD ;
    LM_DC_2ND_CLAMP7_RET_LP : WORD ;
    LM_DC_1ST_CLAMP5_ADV_LP : WORD ;
    LM_DC_1ST_CLAMP5_RET_LP : WORD ;
    SP_WORD68 : WORD ;
    SP_WORD69 : WORD ;
    SP_WORD70 : WORD ;
    SP_WORD71 : WORD ;
    TL_DC_PIN_UP_LP : WORD ;
    TL_DC_PIN_DOWN_LP : WORD ;
    TL_DC_LATCH1_ADV_LP : WORD ;
    TL_DC_LATCH1_RET_LP : WORD ;
    TL_DC_LATCH2_ADV_LP : WORD ;
    TL_DC_LATCH2_RET_LP : WORD ;
    TL_DC_1ST_CLAMP1_ADV_LP : WORD ;
    TL_DC_1ST_CLAMP1_RET_LP : WORD ;
    TL_DC_1ST_CLAMP2_ADV_LP : WORD ;
    TL_DC_1ST_CLAMP2_RET_LP : WORD ;
    TL_DC_1ST_CLAMP3_ADV_LP : WORD ;
    TL_DC_1ST_CLAMP3_RET_LP : WORD ;
    TL_DC_2ND_CLAMP1_ADV_LP : WORD ;
    TL_DC_2ND_CLAMP1_RET_LP : WORD ;
    TL_DC_2ND_CLAMP2_ADV_LP : WORD ;
    TL_DC_2ND_CLAMP2_RET_LP : WORD ;
    TL_DC_U261_ADV_LP : WORD ;
    TL_DC_U261_RET_LP : WORD ;
    TL_DC_U261_CLAMP_ADV_LP : WORD ;
    TL_DC_U261_CLAMP_RET_LP : WORD ;
    TL_DC_U269_UP_LP : WORD ;
    TL_DC_U269_DOWN_LP : WORD ;
    TL_DC_U269_CLAMP_ADV_LP : WORD ;
    TL_DC_U269_CLAMP_RET_LP : WORD ;
    TL_DC_3RD_CLAMP_ADV_LP : WORD ;
    TL_DC_3RD_CLAMP_RET_LP : WORD ;
    TL_DC_U262_1_UP_LP : WORD ;
    TL_DC_U262_1_DOWN_LP : WORD ;
    TL_DC_U262_1_ADV_LP : WORD ;
    TL_DC_U262_1_RET_LP : WORD ;
    TL_DC_U262_1_CLP_ADV_LP : WORD ;
    TL_DC_U262_1_CLP_RET_LP : WORD ;
    TL_DC_U261_2_CLP_ADV_LP : WORD ;
    TL_DC_U261_2_CLP_RET_LP : WORD ;
    SP_WORD106 : WORD ;
    SP_WORD107 : WORD ;
    SP_WORD108 : WORD ;
    SP_WORD109 : WORD ;
    SP_WORD110 : WORD ;
    SP_WORD111 : WORD ;
   END_STRUCT ;
   S_707 : STRUCT
    M_AUTO_SEL : BOOL ;
    M_MANUAL_SEL : BOOL ;
    M_READY_PB : BOOL ;
    M_AUTO_RUN_PB : BOOL ;
    M_WORK_COMP_SET_PB : BOOL ;
    M_WORK_COMP_RST_PB : BOOL ;
    M_HOME_POS_PB : BOOL ;
    M_TIP_DRESS_PB : BOOL ;
    HOOK_PIN_SEL : BOOL ;
    DAECHA_LOCK_SEL : BOOL ;
    ELE_SEL : BOOL ;
    SPARE12 : BOOL ;
    SPARE13 : BOOL ;
    SPARE14 : BOOL ;
    SPARE15 : BOOL ;
    SPARE16 : BOOL ;
    SPARE17 : BOOL ;
    SPARE18 : BOOL ;
    SPARE19 : BOOL ;
    SPARE20 : BOOL ;
    SPARE21 : BOOL ;
    SPARE22 : BOOL ;
    SPARE23 : BOOL ;
    SPARE24 : BOOL ;
    SPARE25 : BOOL ;
    SPARE26 : BOOL ;
    SPARE27 : BOOL ;
    SPARE28 : BOOL ;
    SPARE29 : BOOL ;
    SPARE30 : BOOL ;
    M_ADV_PB : BOOL ;
    M_RET_PB : BOOL ;
    LM_DC_PIN_SEL : BOOL ;
    LM_DC_1ST_CLAMP1_SEL : BOOL ;
    LM_DC_1ST_CLAMP2_SEL : BOOL ;
    LM_DC_1ST_CLAMP3_SEL : BOOL ;
    LM_DC_1ST_CLAMP4_SEL : BOOL ;
    LM_DC_2ND_CLAMP1_SEL : BOOL ;
    LM_DC_2ND_CLAMP2_SEL : BOOL ;
    LM_DC_2ND_CLAMP3_SEL : BOOL ;
    LM_DC_2ND_CLAMP4_SEL : BOOL ;
    LM_DC_2ND_CLAMP5_SEL : BOOL ;
    LM_DC_DR_STK_PIN_SEL : BOOL ;
    LM_DC_OTR_CLAMP_SEL : BOOL ;
    LM_DC_ASSY_CLAMP_SEL : BOOL ;
    LM_DC_FF_PIN_SEL : BOOL ;
    LM_DC_FF_CLAMP_SEL : BOOL ;
    LM_DC_2ND_CLAMP6_SEL : BOOL ;
    SPARE50 : BOOL ;
    SPARE51 : BOOL ;
    SPARE52 : BOOL ;
    SPARE53 : BOOL ;
    SPARE54 : BOOL ;
    SPARE55 : BOOL ;
    SPARE56 : BOOL ;
    SPARE57 : BOOL ;
    SPARE58 : BOOL ;
    SPARE59 : BOOL ;
    SPARE60 : BOOL ;
    SPARE61 : BOOL ;
    SPARE62 : BOOL ;
    SPARE63 : BOOL ;
    LM_DC_M_ADV_PB : BOOL ;
    LM_DC_M_RET_PB : BOOL ;
    TL_DC_PIN_SEL : BOOL ;
    TL_DC_LATCH1_SEL : BOOL ;
    TL_DC_1ST_CLAMP_SEL : BOOL ;
    TL_DC_2ND_CLAMP_SEL : BOOL ;
    TL_DC_U261_SEL : BOOL ;
    TL_DC_U261_CLAMP_SEL : BOOL ;
    TL_DC_U269_UP_DN_SEL : BOOL ;
    TL_DC_U269_CLAMP_SEL : BOOL ;
    TL_DC_3RD_CLAMP_SEL : BOOL ;
    TL_DC_U262_1_UP_DN_SEL : BOOL ;
    TL_DC_U262_1_SEL : BOOL ;
    TL_DC_U262_1_CLAMP_SEL : BOOL ;
    TL_DC_U261_2_CLAMP_SEL : BOOL ;
    SPARE79 : BOOL ;
    SPARE80 : BOOL ;
    SPARE81 : BOOL ;
    SPARE82 : BOOL ;
    SPARE83 : BOOL ;
    SPARE84 : BOOL ;
    SPARE85 : BOOL ;
    SPARE86 : BOOL ;
    SPARE87 : BOOL ;
    SPARE88 : BOOL ;
    SPARE89 : BOOL ;
    SPARE90 : BOOL ;
    SPARE91 : BOOL ;
    SPARE92 : BOOL ;
    SPARE93 : BOOL ;
    SPARE94 : BOOL ;
    SPARE95 : BOOL ;
    TL_DC_M_ADV_PB : BOOL ;
    TL_DC_M_RET_PB : BOOL ;
    SPARE98 : BOOL ;
    SPARE99 : BOOL ;
    SPARE100 : BOOL ;
    SPARE101 : BOOL ;
    SPARE102 : BOOL ;
    SPARE103 : BOOL ;
    SPARE104 : BOOL ;
    SPARE105 : BOOL ;
    SPARE106 : BOOL ;
    SPARE107 : BOOL ;
    SPARE108 : BOOL ;
    SPARE109 : BOOL ;
    SPARE110 : BOOL ;
    SPARE111 : BOOL ;
    SPARE112 : BOOL ;
    SPARE113 : BOOL ;
    SPARE114 : BOOL ;
    SPARE115 : BOOL ;
    SPARE116 : BOOL ;
    SPARE117 : BOOL ;
    SPARE118 : BOOL ;
    SPARE119 : BOOL ;
    SPARE120 : BOOL ;
    SPARE121 : BOOL ;
    SPARE122 : BOOL ;
    SPARE123 : BOOL ;
    SPARE124 : BOOL ;
    SPARE125 : BOOL ;
    SPARE126 : BOOL ;
    SPARE127 : BOOL ;
    SPARE128 : BOOL ;
    SPARE129 : BOOL ;
    SPARE130 : BOOL ;
    SPARE131 : BOOL ;
    SPARE132 : BOOL ;
    SPARE133 : BOOL ;
    SPARE134 : BOOL ;
    SPARE135 : BOOL ;
    SPARE136 : BOOL ;
    SPARE137 : BOOL ;
    SPARE138 : BOOL ;
    SPARE139 : BOOL ;
    SPARE140 : BOOL ;
    SPARE141 : BOOL ;
    SPARE142 : BOOL ;
    SPARE143 : BOOL ;
    SPARE144 : BOOL ;
    SPARE145 : BOOL ;
    SPARE146 : BOOL ;
    SPARE147 : BOOL ;
    SPARE148 : BOOL ;
    SPARE149 : BOOL ;
    SPARE150 : BOOL ;
    SPARE151 : BOOL ;
    SPARE152 : BOOL ;
    SPARE153 : BOOL ;
    SPARE154 : BOOL ;
    SPARE155 : BOOL ;
    SPARE156 : BOOL ;
    SPARE157 : BOOL ;
    SPARE158 : BOOL ;
    SPARE159 : BOOL ;
    SPARE160 : BOOL ;
    SPARE161 : BOOL ;
    HOOK_PIN_UP_LP : WORD ;
    HOOK_PIN_DOWN_LP : WORD ;
    DAECHA_LOCK_ADV_LP : WORD ;
    DAECHA_LOCK_RET_LP : WORD ;
    ELE_ADV_LP : WORD ;
    ELE_RET_LP : WORD ;
    AIR_ELE_ADV_LP : WORD ;
    AIR_ELE_RET_LP : WORD ;
    SP_WORD19 : WORD ;
    SP_WORD20 : WORD ;
    LM_DC_PIN_UP_LP : WORD ;
    LM_DC_PIN_DOWN_LP : WORD ;
    LM_DC_1ST_CLAMP1_ADV_LP : WORD ;
    LM_DC_1ST_CLAMP1_RET_LP : WORD ;
    LM_DC_1ST_CLAMP2_ADV_LP : WORD ;
    LM_DC_1ST_CLAMP2_RET_LP : WORD ;
    LM_DC_1ST_CLAMP3_ADV_LP : WORD ;
    LM_DC_1ST_CLAMP3_RET_LP : WORD ;
    LM_DC_1ST_CLAMP4_ADV_LP : WORD ;
    LM_DC_1ST_CLAMP4_RET_LP : WORD ;
    LM_DC_2ND_CLAMP1_ADV_LP : WORD ;
    LM_DC_2ND_CLAMP1_RET_LP : WORD ;
    LM_DC_2ND_CLAMP2_ADV_LP : WORD ;
    LM_DC_2ND_CLAMP2_RET_LP : WORD ;
    LM_DC_2ND_CLAMP3_ADV_LP : WORD ;
    LM_DC_2ND_CLAMP3_RET_LP : WORD ;
    LM_DC_2ND_CLAMP4_ADV_LP : WORD ;
    LM_DC_2ND_CLAMP4_RET_LP : WORD ;
    LM_DC_2ND_CLAMP5_ADV_LP : WORD ;
    LM_DC_2ND_CLAMP5_RET_LP : WORD ;
    LM_DC_DR_STK_PIN_UP_LP : WORD ;
    LM_DC_DR_STK_PIN_DOWN_LP : WORD ;
    LM_DC_OTR_CLAMP_ADV_LP : WORD ;
    LM_DC_OTR_CLAMP_RET_LP : WORD ;
    LM_DC_ASSY_CLAMP_ADV_LP : WORD ;
    LM_DC_ASSY_CLAMP_RET_LP : WORD ;
    LM_DC_FF_PIN_UP_LP : WORD ;
    LM_DC_FF_PIN_DOWN_LP : WORD ;
    LM_DC_FF_CLAMP_ADV_LP : WORD ;
    LM_DC_FF_CLAMP_RET_LP : WORD ;
    LM_DC_2ND_CLAMP6_ADV_LP : WORD ;
    LM_DC_2ND_CLAMP6_RET_LP : WORD ;
    LM_DC_2ND_CLAMP7_ADV_LP : WORD ;
    LM_DC_2ND_CLAMP7_RET_LP : WORD ;
    LM_DC_1ST_CLAMP5_ADV_LP : WORD ;
    LM_DC_1ST_CLAMP5_RET_LP : WORD ;
    SP_WORD68 : WORD ;
    SP_WORD69 : WORD ;
    SP_WORD70 : WORD ;
    SP_WORD71 : WORD ;
    TL_DC_PIN_UP_LP : WORD ;
    TL_DC_PIN_DOWN_LP : WORD ;
    TL_DC_LATCH1_ADV_LP : WORD ;
    TL_DC_LATCH1_RET_LP : WORD ;
    TL_DC_LATCH2_ADV_LP : WORD ;
    TL_DC_LATCH2_RET_LP : WORD ;
    TL_DC_1ST_CLAMP1_ADV_LP : WORD ;
    TL_DC_1ST_CLAMP1_RET_LP : WORD ;
    TL_DC_1ST_CLAMP2_ADV_LP : WORD ;
    TL_DC_1ST_CLAMP2_RET_LP : WORD ;
    TL_DC_1ST_CLAMP3_ADV_LP : WORD ;
    TL_DC_1ST_CLAMP3_RET_LP : WORD ;
    TL_DC_2ND_CLAMP1_ADV_LP : WORD ;
    TL_DC_2ND_CLAMP1_RET_LP : WORD ;
    TL_DC_2ND_CLAMP2_ADV_LP : WORD ;
    TL_DC_2ND_CLAMP2_RET_LP : WORD ;
    TL_DC_U261_ADV_LP : WORD ;
    TL_DC_U261_RET_LP : WORD ;
    TL_DC_U261_CLAMP_ADV_LP : WORD ;
    TL_DC_U261_CLAMP_RET_LP : WORD ;
    TL_DC_U269_UP_LP : WORD ;
    TL_DC_U269_DOWN_LP : WORD ;
    TL_DC_U269_CLAMP_ADV_LP : WORD ;
    TL_DC_U269_CLAMP_RET_LP : WORD ;
    TL_DC_3RD_CLAMP_ADV_LP : WORD ;
    TL_DC_3RD_CLAMP_RET_LP : WORD ;
    TL_DC_U262_1_UP_LP : WORD ;
    TL_DC_U262_1_DOWN_LP : WORD ;
    TL_DC_U262_1_ADV_LP : WORD ;
    TL_DC_U262_1_RET_LP : WORD ;
    TL_DC_U262_1_CLP_ADV_LP : WORD ;
    TL_DC_U262_1_CLP_RET_LP : WORD ;
    TL_DC_U261_2_CLP_ADV_LP : WORD ;
    TL_DC_U261_2_CLP_RET_LP : WORD ;
    SP_WORD106 : WORD ;
    SP_WORD107 : WORD ;
    SP_WORD108 : WORD ;
    SP_WORD109 : WORD ;
    SP_WORD110 : WORD ;
    SP_WORD111 : WORD ;
   END_STRUCT ;
   S_708 : STRUCT
    M_AUTO_SEL : BOOL ;
    M_MANUAL_SEL : BOOL ;
    M_READY_PB : BOOL ;
    M_AUTO_RUN_PB : BOOL ;
    M_WORK_COMP_SET_PB : BOOL ;
    M_WORK_COMP_RST_PB : BOOL ;
    M_HOME_POS_PB : BOOL ;
    M_708_L_R_BT_ERR_RST : BOOL ;
    HOOK_PIN_SEL : BOOL ;
    EJECT_SEL : BOOL ;
    SAFETY_PIN_SEL : BOOL ;
    DAECHA_OUT_SEL : BOOL ;
    ELE_UP_DN_SEL : BOOL ;
    ELE_ADV_RET_SEL : BOOL ;
    SPARE15 : BOOL ;
    SPARE16 : BOOL ;
    SPARE17 : BOOL ;
    SPARE18 : BOOL ;
    SPARE19 : BOOL ;
    SPARE20 : BOOL ;
    SPARE21 : BOOL ;
    SPARE22 : BOOL ;
    SPARE23 : BOOL ;
    SPARE24 : BOOL ;
    SPARE25 : BOOL ;
    SPARE26 : BOOL ;
    SPARE27 : BOOL ;
    SPARE28 : BOOL ;
    SPARE29 : BOOL ;
    SPARE30 : BOOL ;
    M_ADV_PB : BOOL ;
    M_RET_PB : BOOL ;
    LM_DC_PIN_SEL : BOOL ;
    LM_DC_1ST_CLAMP1_SEL : BOOL ;
    LM_DC_1ST_CLAMP2_SEL : BOOL ;
    LM_DC_1ST_CLAMP3_SEL : BOOL ;
    LM_DC_1ST_CLAMP4_SEL : BOOL ;
    LM_DC_2ND_CLAMP1_SEL : BOOL ;
    LM_DC_2ND_CLAMP2_SEL : BOOL ;
    LM_DC_2ND_CLAMP3_SEL : BOOL ;
    LM_DC_2ND_CLAMP4_SEL : BOOL ;
    LM_DC_2ND_CLAMP5_SEL : BOOL ;
    LM_DC_DR_STK_PIN_SEL : BOOL ;
    LM_DC_OTR_CLAMP_SEL : BOOL ;
    LM_DC_ASSY_CLAMP_SEL : BOOL ;
    LM_DC_FF_PIN_SEL : BOOL ;
    LM_DC_FF_CLAMP_SEL : BOOL ;
    LM_DC_2ND_CLAMP6_SEL : BOOL ;
    SPARE50 : BOOL ;
    SPARE51 : BOOL ;
    SPARE52 : BOOL ;
    SPARE53 : BOOL ;
    SPARE54 : BOOL ;
    SPARE55 : BOOL ;
    SPARE56 : BOOL ;
    SPARE57 : BOOL ;
    SPARE58 : BOOL ;
    SPARE59 : BOOL ;
    SPARE60 : BOOL ;
    SPARE61 : BOOL ;
    SPARE62 : BOOL ;
    SPARE63 : BOOL ;
    LM_DC_M_ADV_PB : BOOL ;
    LM_DC_M_RET_PB : BOOL ;
    TL_DC_PIN_SEL : BOOL ;
    TL_DC_LATCH1_SEL : BOOL ;
    TL_DC_1ST_CLAMP_SEL : BOOL ;
    TL_DC_2ND_CLAMP_SEL : BOOL ;
    TL_DC_U261_SEL : BOOL ;
    TL_DC_U261_CLAMP_SEL : BOOL ;
    TL_DC_U269_UP_DN_SEL : BOOL ;
    TL_DC_U269_CLAMP_SEL : BOOL ;
    TL_DC_3RD_CLAMP_SEL : BOOL ;
    TL_DC_U262_1_UP_DN_SEL : BOOL ;
    TL_DC_U262_1_SEL : BOOL ;
    TL_DC_U262_1_CLAMP_SEL : BOOL ;
    TL_DC_U261_2_CLAMP_SEL : BOOL ;
    SPARE79 : BOOL ;
    SPARE80 : BOOL ;
    SPARE81 : BOOL ;
    SPARE82 : BOOL ;
    SPARE83 : BOOL ;
    SPARE84 : BOOL ;
    SPARE85 : BOOL ;
    SPARE86 : BOOL ;
    SPARE87 : BOOL ;
    SPARE88 : BOOL ;
    SPARE89 : BOOL ;
    SPARE90 : BOOL ;
    SPARE91 : BOOL ;
    SPARE92 : BOOL ;
    SPARE93 : BOOL ;
    SPARE94 : BOOL ;
    SPARE95 : BOOL ;
    TL_DC_M_ADV_PB : BOOL ;
    TL_DC_M_RET_PB : BOOL ;
    SPARE98 : BOOL ;
    SPARE99 : BOOL ;
    SPARE100 : BOOL ;
    SPARE101 : BOOL ;
    SPARE102 : BOOL ;
    SPARE103 : BOOL ;
    SPARE104 : BOOL ;
    SPARE105 : BOOL ;
    SPARE106 : BOOL ;
    SPARE107 : BOOL ;
    SPARE108 : BOOL ;
    SPARE109 : BOOL ;
    SPARE110 : BOOL ;
    SPARE111 : BOOL ;
    SPARE112 : BOOL ;
    SPARE113 : BOOL ;
    SPARE114 : BOOL ;
    SPARE115 : BOOL ;
    SPARE116 : BOOL ;
    SPARE117 : BOOL ;
    SPARE118 : BOOL ;
    SPARE119 : BOOL ;
    SPARE120 : BOOL ;
    SPARE121 : BOOL ;
    SPARE122 : BOOL ;
    SPARE123 : BOOL ;
    SPARE124 : BOOL ;
    SPARE125 : BOOL ;
    SPARE126 : BOOL ;
    SPARE127 : BOOL ;
    SPARE128 : BOOL ;
    SPARE129 : BOOL ;
    ELE_AR_ADV_LP : WORD ;
    ELE_AR_RET_LP : WORD ;
    HOOK_PIN_UP_LP : WORD ;
    HOOK_PIN_DOWN_LP : WORD ;
    EJECT_UP_LP : WORD ;
    EJECT_DOWN_LP : WORD ;
    SAFETY_PIN_UP_LP : WORD ;
    SAFETY_PIN_UDOWN_LP : WORD ;
    DAECHA_OUT_ADV_LP : WORD ;
    DAECHA_OUT_RET_LP : WORD ;
    ELE_UD_UP_LP : WORD ;
    ELE_UD_DOWN_LP : WORD ;
    LM_DC_PIN_UP_LP : WORD ;
    LM_DC_PIN_DOWN_LP : WORD ;
    LM_DC_1ST_CLAMP1_ADV_LP : WORD ;
    LM_DC_1ST_CLAMP1_RET_LP : WORD ;
    LM_DC_1ST_CLAMP2_ADV_LP : WORD ;
    LM_DC_1ST_CLAMP2_RET_LP : WORD ;
    LM_DC_1ST_CLAMP3_ADV_LP : WORD ;
    LM_DC_1ST_CLAMP3_RET_LP : WORD ;
    LM_DC_1ST_CLAMP4_ADV_LP : WORD ;
    LM_DC_1ST_CLAMP4_RET_LP : WORD ;
    LM_DC_2ND_CLAMP1_ADV_LP : WORD ;
    LM_DC_2ND_CLAMP1_RET_LP : WORD ;
    LM_DC_2ND_CLAMP2_ADV_LP : WORD ;
    LM_DC_2ND_CLAMP2_RET_LP : WORD ;
    LM_DC_2ND_CLAMP3_ADV_LP : WORD ;
    LM_DC_2ND_CLAMP3_RET_LP : WORD ;
    LM_DC_2ND_CLAMP4_ADV_LP : WORD ;
    LM_DC_2ND_CLAMP4_RET_LP : WORD ;
    LM_DC_2ND_CLAMP5_ADV_LP : WORD ;
    LM_DC_2ND_CLAMP5_RET_LP : WORD ;
    LM_DC_DR_STK_PIN_UP_LP : WORD ;
    LM_DC_DR_STK_PIN_DOWN_LP : WORD ;
    LM_DC_OTR_CLAMP_ADV_LP : WORD ;
    LM_DC_OTR_CLAMP_RET_LP : WORD ;
    LM_DC_ASSY_CLAMP_ADV_LP : WORD ;
    LM_DC_ASSY_CLAMP_RET_LP : WORD ;
    LM_DC_FF_PIN_UP_LP : WORD ;
    LM_DC_FF_PIN_DOWN_LP : WORD ;
    LM_DC_FF_CLAMP_ADV_LP : WORD ;
    LM_DC_FF_CLAMP_RET_LP : WORD ;
    LM_DC_2ND_CLAMP6_ADV_LP : WORD ;
    LM_DC_2ND_CLAMP6_RET_LP : WORD ;
    LM_DC_2ND_CLAMP7_ADV_LP : WORD ;
    LM_DC_2ND_CLAMP7_RET_LP : WORD ;
    LM_DC_1ST_CLAMP5_ADV_LP : WORD ;
    LM_DC_1ST_CLAMP5_RET_LP : WORD ;
    SP_WORD68 : WORD ;
    SP_WORD69 : WORD ;
    SP_WORD70 : WORD ;
    SP_WORD71 : WORD ;
    TL_DC_PIN_UP_LP : WORD ;
    TL_DC_PIN_DOWN_LP : WORD ;
    TL_DC_LATCH1_ADV_LP : WORD ;
    TL_DC_LATCH1_RET_LP : WORD ;
    TL_DC_LATCH2_ADV_LP : WORD ;
    TL_DC_LATCH2_RET_LP : WORD ;
    TL_DC_1ST_CLAMP1_ADV_LP : WORD ;
    TL_DC_1ST_CLAMP1_RET_LP : WORD ;
    TL_DC_1ST_CLAMP2_ADV_LP : WORD ;
    TL_DC_1ST_CLAMP2_RET_LP : WORD ;
    TL_DC_1ST_CLAMP3_ADV_LP : WORD ;
    TL_DC_1ST_CLAMP3_RET_LP : WORD ;
    TL_DC_2ND_CLAMP1_ADV_LP : WORD ;
    TL_DC_2ND_CLAMP1_RET_LP : WORD ;
    TL_DC_2ND_CLAMP2_ADV_LP : WORD ;
    TL_DC_2ND_CLAMP2_RET_LP : WORD ;
    TL_DC_U261_ADV_LP : WORD ;
    TL_DC_U261_RET_LP : WORD ;
    TL_DC_U261_CLAMP_ADV_LP : WORD ;
    TL_DC_U261_CLAMP_RET_LP : WORD ;
    TL_DC_U269_UP_LP : WORD ;
    TL_DC_U269_DOWN_LP : WORD ;
    TL_DC_U269_CLAMP_ADV_LP : WORD ;
    TL_DC_U269_CLAMP_RET_LP : WORD ;
    TL_DC_3RD_CLAMP_ADV_LP : WORD ;
    TL_DC_3RD_CLAMP_RET_LP : WORD ;
    TL_DC_U262_1_UP_LP : WORD ;
    TL_DC_U262_1_DOWN_LP : WORD ;
    TL_DC_U262_1_ADV_LP : WORD ;
    TL_DC_U262_1_RET_LP : WORD ;
    TL_DC_U262_1_CLP_ADV_LP : WORD ;
    TL_DC_U262_1_CLP_RET_LP : WORD ;
    TL_DC_U261_2_CLP_ADV_LP : WORD ;
    TL_DC_U261_2_CLP_RET_LP : WORD ;
    SP_WORD106 : WORD ;
    SP_WORD107 : WORD ;
    SP_WORD108 : WORD ;
    SP_WORD109 : WORD ;
    AIR_ELE_AR_ADV_LP : WORD ;
    AIR_ELE_AR_RET_LP : WORD ;
   END_STRUCT ;
   S_UPDL : STRUCT
    M_AUTO_SEL : BOOL ;
    M_MANUAL_SEL : BOOL ;
    M_READY_PB : BOOL ;
    M_AUTO_RUN_PB : BOOL ;
    M_WORK_COMP_SET_PB : BOOL ;
    M_WORK_COMP_RST_PB : BOOL ;
    M_HOME_POS_PB : BOOL ;
    SPARE8 : BOOL ;
    DAECHA_CLAMP_SEL : BOOL ;
    ELE_AIR_UP_DN_SEL : BOOL ;
    ELE_AIR_ADV_RET_SEL : BOOL ;
    DAECHA_IN_SEL : BOOL ;
    DAECHA_OUT_SEL : BOOL ;
    LIFT_LOCK_SEL : BOOL ;
    LIFT_UP_DN_SEL : BOOL ;
    SPARE16 : BOOL ;
    SPARE17 : BOOL ;
    SPARE18 : BOOL ;
    SPARE19 : BOOL ;
    SPARE20 : BOOL ;
    SPARE21 : BOOL ;
    SPARE22 : BOOL ;
    SPARE23 : BOOL ;
    SPARE24 : BOOL ;
    SPARE25 : BOOL ;
    SPARE26 : BOOL ;
    SPARE27 : BOOL ;
    SPARE28 : BOOL ;
    SPARE29 : BOOL ;
    SPARE30 : BOOL ;
    M_ADV_PB : BOOL ;
    M_RET_PB : BOOL ;
    SPARE34 : BOOL ;
    SPARE35 : BOOL ;
    SPARE36 : BOOL ;
    SPARE37 : BOOL ;
    SPARE38 : BOOL ;
    SPARE39 : BOOL ;
    SPARE40 : BOOL ;
    SPARE41 : BOOL ;
    SPARE42 : BOOL ;
    SPARE43 : BOOL ;
    SPARE44 : BOOL ;
    SPARE45 : BOOL ;
    SPARE46 : BOOL ;
    SPARE47 : BOOL ;
    SPARE48 : BOOL ;
    SPARE49 : BOOL ;
    SPARE50 : BOOL ;
    SPARE51 : BOOL ;
    SPARE52 : BOOL ;
    SPARE53 : BOOL ;
    SPARE54 : BOOL ;
    SPARE55 : BOOL ;
    SPARE56 : BOOL ;
    SPARE57 : BOOL ;
    SPARE58 : BOOL ;
    SPARE59 : BOOL ;
    SPARE60 : BOOL ;
    SPARE61 : BOOL ;
    SPARE62 : BOOL ;
    SPARE63 : BOOL ;
    SPARE64 : BOOL ;
    SPARE65 : BOOL ;
    SPARE66 : BOOL ;
    SPARE67 : BOOL ;
    SPARE68 : BOOL ;
    SPARE69 : BOOL ;
    SPARE70 : BOOL ;
    SPARE71 : BOOL ;
    SPARE72 : BOOL ;
    SPARE73 : BOOL ;
    SPARE74 : BOOL ;
    SPARE75 : BOOL ;
    SPARE76 : BOOL ;
    SPARE77 : BOOL ;
    SPARE78 : BOOL ;
    SPARE79 : BOOL ;
    SPARE80 : BOOL ;
    SPARE81 : BOOL ;
    SPARE82 : BOOL ;
    SPARE83 : BOOL ;
    SPARE84 : BOOL ;
    SPARE85 : BOOL ;
    SPARE86 : BOOL ;
    SPARE87 : BOOL ;
    SPARE88 : BOOL ;
    SPARE89 : BOOL ;
    SPARE90 : BOOL ;
    SPARE91 : BOOL ;
    SPARE92 : BOOL ;
    SPARE93 : BOOL ;
    SPARE94 : BOOL ;
    SPARE95 : BOOL ;
    SPARE96 : BOOL ;
    SPARE97 : BOOL ;
    SPARE98 : BOOL ;
    SPARE99 : BOOL ;
    SPARE100 : BOOL ;
    SPARE101 : BOOL ;
    SPARE102 : BOOL ;
    SPARE103 : BOOL ;
    SPARE104 : BOOL ;
    SPARE105 : BOOL ;
    SPARE106 : BOOL ;
    SPARE107 : BOOL ;
    SPARE108 : BOOL ;
    SPARE109 : BOOL ;
    SPARE110 : BOOL ;
    SPARE111 : BOOL ;
    SPARE112 : BOOL ;
    SPARE113 : BOOL ;
    SPARE114 : BOOL ;
    SPARE115 : BOOL ;
    SPARE116 : BOOL ;
    SPARE117 : BOOL ;
    SPARE118 : BOOL ;
    SPARE119 : BOOL ;
    SPARE120 : BOOL ;
    SPARE121 : BOOL ;
    SPARE122 : BOOL ;
    SPARE123 : BOOL ;
    SPARE124 : BOOL ;
    SPARE125 : BOOL ;
    SPARE126 : BOOL ;
    SPARE127 : BOOL ;
    SPARE128 : BOOL ;
    SPARE129 : BOOL ;
    SPARE130 : BOOL ;
    SPARE131 : BOOL ;
    SPARE132 : BOOL ;
    SPARE133 : BOOL ;
    SPARE134 : BOOL ;
    SPARE135 : BOOL ;
    SPARE136 : BOOL ;
    SPARE137 : BOOL ;
    SPARE138 : BOOL ;
    SPARE139 : BOOL ;
    SPARE140 : BOOL ;
    SPARE141 : BOOL ;
    SPARE142 : BOOL ;
    SPARE143 : BOOL ;
    SPARE144 : BOOL ;
    SPARE145 : BOOL ;
    SPARE146 : BOOL ;
    SPARE147 : BOOL ;
    SPARE148 : BOOL ;
    SPARE149 : BOOL ;
    SPARE150 : BOOL ;
    SPARE151 : BOOL ;
    SPARE152 : BOOL ;
    SPARE153 : BOOL ;
    SPARE154 : BOOL ;
    SPARE155 : BOOL ;
    SPARE156 : BOOL ;
    SPARE157 : BOOL ;
    SPARE158 : BOOL ;
    SPARE159 : BOOL ;
    SPARE160 : BOOL ;
    SPARE161 : BOOL ;
    DAECHA_CLAMP_ADV_LP : WORD ;
    DAECHA_CLAMP_RET_LP : WORD ;
    ELE_AIR_UP_DN_UP_LP : WORD ;
    ELE_AIR_UP_DN_DOWN_LP : WORD ;
    ELE_AIR_ADV_RET_ADV_LP : WORD ;
    ELE_AIR_ADV_RET_RET_LP : WORD ;
    DAECHA_IN_ADV_LP : WORD ;
    DAECHA_IN_RET_LP : WORD ;
    DAECHA_OUT_ADV_LP : WORD ;
    DAECHA_OUT_RET_LP : WORD ;
    LIFT_LOCL_ADV_LP : WORD ;
    LIFT_LOCL_RET_LP : WORD ;
    LIFT_UP_DN_UP_LP : WORD ;
    LIFT_UP_DN_DOWN_LP : WORD ;
    SP_WORD25 : WORD ;
    SP_WORD26 : WORD ;
    SP_WORD27 : WORD ;
    SP_WORD28 : WORD ;
    SP_WORD29 : WORD ;
    SP_WORD30 : WORD ;
    SP_WORD31 : WORD ;
    SP_WORD32 : WORD ;
    SP_WORD33 : WORD ;
    SP_WORD34 : WORD ;
    SP_WORD35 : WORD ;
    SP_WORD36 : WORD ;
    SP_WORD37 : WORD ;
    SP_WORD38 : WORD ;
    SP_WORD39 : WORD ;
    SP_WORD40 : WORD ;
    SP_WORD41 : WORD ;
    SP_WORD42 : WORD ;
    SP_WORD43 : WORD ;
    SP_WORD44 : WORD ;
    SP_WORD45 : WORD ;
    SP_WORD46 : WORD ;
    SP_WORD47 : WORD ;
    SP_WORD49 : WORD ;
    SP_WORD50 : WORD ;
    SP_WORD51 : WORD ;
    SP_WORD52 : WORD ;
    SP_WORD53 : WORD ;
    SP_WORD54 : WORD ;
    SP_WORD55 : WORD ;
    SP_WORD56 : WORD ;
    SP_WORD57 : WORD ;
    SP_WORD58 : WORD ;
    SP_WORD59 : WORD ;
    SP_WORD60 : WORD ;
    SP_WORD61 : WORD ;
    SP_WORD62 : WORD ;
    SP_WORD63 : WORD ;
    SP_WORD64 : WORD ;
    SP_WORD65 : WORD ;
    SP_WORD66 : WORD ;
    SP_WORD67 : WORD ;
    SP_WORD68 : WORD ;
    SP_WORD69 : WORD ;
    SP_WORD70 : WORD ;
    SP_WORD71 : WORD ;
    SP_WORD72 : WORD ;
    SP_WORD73 : WORD ;
    SP_WORD74 : WORD ;
    SP_WORD75 : WORD ;
    SP_WORD76 : WORD ;
    SP_WORD77 : WORD ;
    SP_WORD78 : WORD ;
    SP_WORD79 : WORD ;
    SP_WORD80 : WORD ;
    SP_WORD81 : WORD ;
    SP_WORD82 : WORD ;
    SP_WORD83 : WORD ;
    SP_WORD84 : WORD ;
    SP_WORD85 : WORD ;
    SP_WORD86 : WORD ;
    SP_WORD87 : WORD ;
    SP_WORD88 : WORD ;
    SP_WORD89 : WORD ;
    SP_WORD90 : WORD ;
    SP_WORD91 : WORD ;
    SP_WORD92 : WORD ;
    SP_WORD93 : WORD ;
    SP_WORD94 : WORD ;
    SP_WORD95 : WORD ;
    SP_WORD96 : WORD ;
    SP_WORD97 : WORD ;
    SP_WORD98 : WORD ;
    SP_WORD99 : WORD ;
    SP_WORD100 : WORD ;
    SP_WORD101 : WORD ;
   END_STRUCT ;
  END_STRUCT ;
BEGIN
   S_705.M_AUTO_SEL := FALSE;
   S_705.M_MANUAL_SEL := FALSE;
   S_705.M_READY_PB := FALSE;
   S_705.M_AUTO_RUN_PB := FALSE;
   S_705.M_WORK_COMP_SET_PB := FALSE;
   S_705.M_WORK_COMP_RST_PB := FALSE;
   S_705.M_HOME_POS_PB := FALSE;
   S_705.M_TIP_DRESS_PB := FALSE;
   S_705.HOOK_PIN_SEL := FALSE;
   S_705.DAECHA_LOCK_SEL := FALSE;
   S_705.ELE_SEL := FALSE;
   S_705.AIR_ELE_SEL := FALSE;
   S_705.SPARE13 := FALSE;
   S_705.SPARE14 := FALSE;
   S_705.SPARE15 := FALSE;
   S_705.SPARE16 := FALSE;
   S_705.SPARE17 := FALSE;
   S_705.SPARE18 := FALSE;
   S_705.SPARE19 := FALSE;
   S_705.SPARE20 := FALSE;
   S_705.SPARE21 := FALSE;
   S_705.SPARE22 := FALSE;
   S_705.SPARE23 := FALSE;
   S_705.SPARE24 := FALSE;
   S_705.SPARE25 := FALSE;
   S_705.SPARE26 := FALSE;
   S_705.SPARE27 := FALSE;
   S_705.SPARE28 := FALSE;
   S_705.SPARE29 := FALSE;
   S_705.SPARE30 := FALSE;
   S_705.M_ADV_PB := FALSE;
   S_705.M_RET_PB := FALSE;
   S_705.LM_DC_PIN_SEL := FALSE;
   S_705.LM_DC_1ST_CLAMP1_SEL := FALSE;
   S_705.LM_DC_1ST_CLAMP2_SEL := FALSE;
   S_705.LM_DC_1ST_CLAMP3_SEL := FALSE;
   S_705.LM_DC_1ST_CLAMP4_SEL := FALSE;
   S_705.LM_DC_2ND_CLAMP1_SEL := FALSE;
   S_705.LM_DC_2ND_CLAMP2_SEL := FALSE;
   S_705.LM_DC_2ND_CLAMP3_SEL := FALSE;
   S_705.LM_DC_2ND_CLAMP4_SEL := FALSE;
   S_705.LM_DC_2ND_CLAMP5_SEL := FALSE;
   S_705.LM_DC_DR_STK_PIN_SEL := FALSE;
   S_705.LM_DC_OTR_CLAMP_SEL := FALSE;
   S_705.LM_DC_ASSY_CLAMP_SEL := FALSE;
   S_705.LM_DC_FF_PIN_SEL := FALSE;
   S_705.LM_DC_FF_CLAMP_SEL := FALSE;
   S_705.LM_DC_2ND_CLAMP6_SEL := FALSE;
   S_705.SPARE50 := FALSE;
   S_705.SPARE51 := FALSE;
   S_705.SPARE52 := FALSE;
   S_705.SPARE53 := FALSE;
   S_705.SPARE54 := FALSE;
   S_705.SPARE55 := FALSE;
   S_705.SPARE56 := FALSE;
   S_705.SPARE57 := FALSE;
   S_705.SPARE58 := FALSE;
   S_705.SPARE59 := FALSE;
   S_705.SPARE60 := FALSE;
   S_705.SPARE61 := FALSE;
   S_705.SPARE62 := FALSE;
   S_705.SPARE63 := FALSE;
   S_705.LM_DC_M_ADV_PB := FALSE;
   S_705.LM_DC_M_RET_PB := FALSE;
   S_705.TL_DC_PIN_SEL := FALSE;
   S_705.TL_DC_LATCH1_SEL := FALSE;
   S_705.TL_DC_1ST_CLAMP_SEL := FALSE;
   S_705.TL_DC_2ND_CLAMP_SEL := FALSE;
   S_705.TL_DC_U261_SEL := FALSE;
   S_705.TL_DC_U261_CLAMP_SEL := FALSE;
   S_705.TL_DC_U269_UP_DN_SEL := FALSE;
   S_705.TL_DC_U269_CLAMP_SEL := FALSE;
   S_705.TL_DC_3RD_CLAMP_SEL := FALSE;
   S_705.TL_DC_U262_1_UP_DN_SEL := FALSE;
   S_705.TL_DC_U262_1_SEL := FALSE;
   S_705.TL_DC_U262_1_CLAMP_SEL := FALSE;
   S_705.TL_DC_U261_2_CLAMP_SEL := FALSE;
   S_705.SPARE79 := FALSE;
   S_705.SPARE80 := FALSE;
   S_705.SPARE81 := FALSE;
   S_705.SPARE82 := FALSE;
   S_705.SPARE83 := FALSE;
   S_705.SPARE84 := FALSE;
   S_705.SPARE85 := FALSE;
   S_705.SPARE86 := FALSE;
   S_705.SPARE87 := FALSE;
   S_705.SPARE88 := FALSE;
   S_705.SPARE89 := FALSE;
   S_705.SPARE90 := FALSE;
   S_705.SPARE91 := FALSE;
   S_705.SPARE92 := FALSE;
   S_705.SPARE93 := FALSE;
   S_705.SPARE94 := FALSE;
   S_705.SPARE95 := FALSE;
   S_705.TL_DC_M_ADV_PB := FALSE;
   S_705.TL_DC_M_RET_PB := FALSE;
   S_705.SPARE98 := FALSE;
   S_705.SPARE99 := FALSE;
   S_705.SPARE100 := FALSE;
   S_705.SPARE101 := FALSE;
   S_705.SPARE102 := FALSE;
   S_705.SPARE103 := FALSE;
   S_705.SPARE104 := FALSE;
   S_705.SPARE105 := FALSE;
   S_705.SPARE106 := FALSE;
   S_705.SPARE107 := FALSE;
   S_705.SPARE108 := FALSE;
   S_705.SPARE109 := FALSE;
   S_705.SPARE110 := FALSE;
   S_705.SPARE111 := FALSE;
   S_705.SPARE112 := FALSE;
   S_705.SPARE113 := FALSE;
   S_705.SPARE114 := FALSE;
   S_705.SPARE115 := FALSE;
   S_705.SPARE116 := FALSE;
   S_705.SPARE117 := FALSE;
   S_705.SPARE118 := FALSE;
   S_705.SPARE119 := FALSE;
   S_705.SPARE120 := FALSE;
   S_705.SPARE121 := FALSE;
   S_705.SPARE122 := FALSE;
   S_705.SPARE123 := FALSE;
   S_705.SPARE124 := FALSE;
   S_705.SPARE125 := FALSE;
   S_705.SPARE126 := FALSE;
   S_705.SPARE127 := FALSE;
   S_705.SPARE128 := FALSE;
   S_705.SPARE129 := FALSE;
   S_705.SPARE130 := FALSE;
   S_705.SPARE131 := FALSE;
   S_705.SPARE132 := FALSE;
   S_705.SPARE133 := FALSE;
   S_705.SPARE134 := FALSE;
   S_705.SPARE135 := FALSE;
   S_705.SPARE136 := FALSE;
   S_705.SPARE137 := FALSE;
   S_705.SPARE138 := FALSE;
   S_705.SPARE139 := FALSE;
   S_705.SPARE140 := FALSE;
   S_705.SPARE141 := FALSE;
   S_705.SPARE142 := FALSE;
   S_705.SPARE143 := FALSE;
   S_705.SPARE144 := FALSE;
   S_705.SPARE145 := FALSE;
   S_705.SPARE146 := FALSE;
   S_705.SPARE147 := FALSE;
   S_705.SPARE148 := FALSE;
   S_705.SPARE149 := FALSE;
   S_705.SPARE150 := FALSE;
   S_705.SPARE151 := FALSE;
   S_705.SPARE152 := FALSE;
   S_705.SPARE153 := FALSE;
   S_705.SPARE154 := FALSE;
   S_705.SPARE155 := FALSE;
   S_705.SPARE156 := FALSE;
   S_705.SPARE157 := FALSE;
   S_705.SPARE158 := FALSE;
   S_705.SPARE159 := FALSE;
   S_705.SPARE160 := FALSE;
   S_705.S705_R2_R3_WORK_COMP_SET := FALSE;
   S_705.HOOK_PIN_UP_LP := W#16#0;
   S_705.HOOK_PIN_DOWN_LP := W#16#300;
   S_705.DAECHA_LOCK_ADV_LP := W#16#300;
   S_705.DAECHA_LOCK_RET_LP := W#16#0;
   S_705.ELE_ADV_LP := W#16#300;
   S_705.ELE_RET_LP := W#16#0;
   S_705.AIR_ELE_ADV_LP := W#16#300;
   S_705.AIR_ELE_RET_LP := W#16#0;
   S_705.SP_WORD19 := W#16#0;
   S_705.SP_WORD20 := W#16#0;
   S_705.LM_DC_PIN_UP_LP := W#16#0;
   S_705.LM_DC_PIN_DOWN_LP := W#16#0;
   S_705.LM_DC_1ST_CLAMP1_ADV_LP := W#16#0;
   S_705.LM_DC_1ST_CLAMP1_RET_LP := W#16#0;
   S_705.LM_DC_1ST_CLAMP2_ADV_LP := W#16#0;
   S_705.LM_DC_1ST_CLAMP2_RET_LP := W#16#0;
   S_705.LM_DC_1ST_CLAMP3_ADV_LP := W#16#0;
   S_705.LM_DC_1ST_CLAMP3_RET_LP := W#16#0;
   S_705.LM_DC_1ST_CLAMP4_ADV_LP := W#16#0;
   S_705.LM_DC_1ST_CLAMP4_RET_LP := W#16#0;
   S_705.LM_DC_2ND_CLAMP1_ADV_LP := W#16#0;
   S_705.LM_DC_2ND_CLAMP1_RET_LP := W#16#0;
   S_705.LM_DC_2ND_CLAMP2_ADV_LP := W#16#0;
   S_705.LM_DC_2ND_CLAMP2_RET_LP := W#16#0;
   S_705.LM_DC_2ND_CLAMP3_ADV_LP := W#16#0;
   S_705.LM_DC_2ND_CLAMP3_RET_LP := W#16#0;
   S_705.LM_DC_2ND_CLAMP4_ADV_LP := W#16#0;
   S_705.LM_DC_2ND_CLAMP4_RET_LP := W#16#0;
   S_705.LM_DC_2ND_CLAMP5_ADV_LP := W#16#0;
   S_705.LM_DC_2ND_CLAMP5_RET_LP := W#16#0;
   S_705.LM_DC_DR_STK_PIN_UP_LP := W#16#0;
   S_705.LM_DC_DR_STK_PIN_DOWN_LP := W#16#0;
   S_705.LM_DC_OTR_CLAMP_ADV_LP := W#16#0;
   S_705.LM_DC_OTR_CLAMP_RET_LP := W#16#0;
   S_705.LM_DC_ASSY_CLAMP_ADV_LP := W#16#0;
   S_705.LM_DC_ASSY_CLAMP_RET_LP := W#16#0;
   S_705.LM_DC_FF_PIN_UP_LP := W#16#0;
   S_705.LM_DC_FF_PIN_DOWN_LP := W#16#0;
   S_705.LM_DC_FF_CLAMP_ADV_LP := W#16#0;
   S_705.LM_DC_FF_CLAMP_RET_LP := W#16#0;
   S_705.LM_DC_2ND_CLAMP6_ADV_LP := W#16#0;
   S_705.LM_DC_2ND_CLAMP6_RET_LP := W#16#0;
   S_705.LM_DC_2ND_CLAMP7_ADV_LP := W#16#0;
   S_705.LM_DC_2ND_CLAMP7_RET_LP := W#16#0;
   S_705.LM_DC_1ST_CLAMP5_ADV_LP := W#16#0;
   S_705.LM_DC_1ST_CLAMP5_RET_LP := W#16#0;
   S_705.SP_WORD68 := W#16#0;
   S_705.SP_WORD69 := W#16#0;
   S_705.SP_WORD70 := W#16#0;
   S_705.SP_WORD71 := W#16#0;
   S_705.TL_DC_PIN_UP_LP := W#16#F00;
   S_705.TL_DC_PIN_DOWN_LP := W#16#0;
   S_705.TL_DC_LATCH1_ADV_LP := W#16#0;
   S_705.TL_DC_LATCH1_RET_LP := W#16#3F00;
   S_705.TL_DC_LATCH2_ADV_LP := W#16#0;
   S_705.TL_DC_LATCH2_RET_LP := W#16#100;
   S_705.TL_DC_1ST_CLAMP1_ADV_LP := W#16#0;
   S_705.TL_DC_1ST_CLAMP1_RET_LP := W#16#3F00;
   S_705.TL_DC_1ST_CLAMP2_ADV_LP := W#16#0;
   S_705.TL_DC_1ST_CLAMP2_RET_LP := W#16#3F00;
   S_705.TL_DC_1ST_CLAMP3_ADV_LP := W#16#0;
   S_705.TL_DC_1ST_CLAMP3_RET_LP := W#16#F00;
   S_705.TL_DC_2ND_CLAMP1_ADV_LP := W#16#0;
   S_705.TL_DC_2ND_CLAMP1_RET_LP := W#16#3F00;
   S_705.TL_DC_2ND_CLAMP2_ADV_LP := W#16#0;
   S_705.TL_DC_2ND_CLAMP2_RET_LP := W#16#3F00;
   S_705.TL_DC_U261_ADV_LP := W#16#0;
   S_705.TL_DC_U261_RET_LP := W#16#100;
   S_705.TL_DC_U261_CLAMP_ADV_LP := W#16#0;
   S_705.TL_DC_U261_CLAMP_RET_LP := W#16#100;
   S_705.TL_DC_U269_UP_LP := W#16#0;
   S_705.TL_DC_U269_DOWN_LP := W#16#300;
   S_705.TL_DC_U269_CLAMP_ADV_LP := W#16#0;
   S_705.TL_DC_U269_CLAMP_RET_LP := W#16#100;
   S_705.TL_DC_3RD_CLAMP_ADV_LP := W#16#0;
   S_705.TL_DC_3RD_CLAMP_RET_LP := W#16#300;
   S_705.TL_DC_U262_1_UP_LP := W#16#0;
   S_705.TL_DC_U262_1_DOWN_LP := W#16#300;
   S_705.TL_DC_U262_1_ADV_LP := W#16#0;
   S_705.TL_DC_U262_1_RET_LP := W#16#300;
   S_705.TL_DC_U262_1_CLP_ADV_LP := W#16#0;
   S_705.TL_DC_U262_1_CLP_RET_LP := W#16#300;
   S_705.TL_DC_U261_2_CLP_ADV_LP := W#16#0;
   S_705.TL_DC_U261_2_CLP_RET_LP := W#16#300;
   S_705.SP_WORD106 := W#16#0;
   S_705.SP_WORD107 := W#16#0;
   S_705.SP_WORD108 := W#16#0;
   S_705.SP_WORD109 := W#16#0;
   S_705.SP_WORD110 := W#16#0;
   S_705.SP_WORD111 := W#16#0;
   S_706.M_AUTO_SEL := FALSE;
   S_706.M_MANUAL_SEL := FALSE;
   S_706.M_READY_PB := FALSE;
   S_706.M_AUTO_RUN_PB := FALSE;
   S_706.M_WORK_COMP_SET_PB := FALSE;
   S_706.M_WORK_COMP_RST_PB := FALSE;
   S_706.M_HOME_POS_PB := FALSE;
   S_706.M_TIP_DRESS_PB := FALSE;
   S_706.HOOK_PIN_SEL := FALSE;
   S_706.DAECHA_LOCK_SEL := FALSE;
   S_706.ELE_SEL := FALSE;
   S_706.AIR_ELE_SEL := FALSE;
   S_706.SPARE13 := FALSE;
   S_706.SPARE14 := FALSE;
   S_706.SPARE15 := FALSE;
   S_706.SPARE16 := FALSE;
   S_706.SPARE17 := FALSE;
   S_706.SPARE18 := FALSE;
   S_706.SPARE19 := FALSE;
   S_706.SPARE20 := FALSE;
   S_706.SPARE21 := FALSE;
   S_706.SPARE22 := FALSE;
   S_706.SPARE23 := FALSE;
   S_706.SPARE24 := FALSE;
   S_706.SPARE25 := FALSE;
   S_706.SPARE26 := FALSE;
   S_706.SPARE27 := FALSE;
   S_706.SPARE28 := FALSE;
   S_706.SPARE29 := FALSE;
   S_706.SPARE30 := FALSE;
   S_706.M_ADV_PB := FALSE;
   S_706.M_RET_PB := FALSE;
   S_706.LM_DC_PIN_SEL := FALSE;
   S_706.LM_DC_1ST_CLAMP1_SEL := FALSE;
   S_706.LM_DC_1ST_CLAMP2_SEL := FALSE;
   S_706.LM_DC_1ST_CLAMP3_SEL := FALSE;
   S_706.LM_DC_1ST_CLAMP4_SEL := FALSE;
   S_706.LM_DC_2ND_CLAMP1_SEL := FALSE;
   S_706.LM_DC_2ND_CLAMP2_SEL := FALSE;
   S_706.LM_DC_2ND_CLAMP3_SEL := FALSE;
   S_706.LM_DC_2ND_CLAMP4_SEL := FALSE;
   S_706.LM_DC_2ND_CLAMP5_SEL := FALSE;
   S_706.LM_DC_DR_STK_PIN_SEL := FALSE;
   S_706.LM_DC_OTR_CLAMP_SEL := FALSE;
   S_706.LM_DC_ASSY_CLAMP_SEL := FALSE;
   S_706.LM_DC_FF_PIN_SEL := FALSE;
   S_706.LM_DC_FF_CLAMP_SEL := FALSE;
   S_706.LM_DC_2ND_CLAMP6_SEL := FALSE;
   S_706.SPARE50 := FALSE;
   S_706.SPARE51 := FALSE;
   S_706.SPARE52 := FALSE;
   S_706.SPARE53 := FALSE;
   S_706.SPARE54 := FALSE;
   S_706.SPARE55 := FALSE;
   S_706.SPARE56 := FALSE;
   S_706.SPARE57 := FALSE;
   S_706.SPARE58 := FALSE;
   S_706.SPARE59 := FALSE;
   S_706.SPARE60 := FALSE;
   S_706.SPARE61 := FALSE;
   S_706.SPARE62 := FALSE;
   S_706.SPARE63 := FALSE;
   S_706.LM_DC_M_ADV_PB := FALSE;
   S_706.LM_DC_M_RET_PB := FALSE;
   S_706.TL_DC_PIN_SEL := FALSE;
   S_706.TL_DC_LATCH1_SEL := FALSE;
   S_706.TL_DC_1ST_CLAMP_SEL := FALSE;
   S_706.TL_DC_2ND_CLAMP_SEL := FALSE;
   S_706.TL_DC_U261_SEL := FALSE;
   S_706.TL_DC_U261_CLAMP_SEL := FALSE;
   S_706.TL_DC_U269_UP_DN_SEL := FALSE;
   S_706.TL_DC_U269_CLAMP_SEL := FALSE;
   S_706.TL_DC_3RD_CLAMP_SEL := FALSE;
   S_706.TL_DC_U262_1_UP_DN_SEL := FALSE;
   S_706.TL_DC_U262_1_SEL := FALSE;
   S_706.TL_DC_U262_1_CLAMP_SEL := FALSE;
   S_706.TL_DC_U261_2_CLAMP_SEL := FALSE;
   S_706.SPARE79 := FALSE;
   S_706.SPARE80 := FALSE;
   S_706.SPARE81 := FALSE;
   S_706.SPARE82 := FALSE;
   S_706.SPARE83 := FALSE;
   S_706.SPARE84 := FALSE;
   S_706.SPARE85 := FALSE;
   S_706.SPARE86 := FALSE;
   S_706.SPARE87 := FALSE;
   S_706.SPARE88 := FALSE;
   S_706.SPARE89 := FALSE;
   S_706.SPARE90 := FALSE;
   S_706.SPARE91 := FALSE;
   S_706.SPARE92 := FALSE;
   S_706.SPARE93 := FALSE;
   S_706.SPARE94 := FALSE;
   S_706.SPARE95 := FALSE;
   S_706.TL_DC_M_ADV_PB := FALSE;
   S_706.TL_DC_M_RET_PB := FALSE;
   S_706.SPARE98 := FALSE;
   S_706.SPARE99 := FALSE;
   S_706.SPARE100 := FALSE;
   S_706.SPARE101 := FALSE;
   S_706.SPARE102 := FALSE;
   S_706.SPARE103 := FALSE;
   S_706.SPARE104 := FALSE;
   S_706.SPARE105 := FALSE;
   S_706.SPARE106 := FALSE;
   S_706.SPARE107 := FALSE;
   S_706.SPARE108 := FALSE;
   S_706.SPARE109 := FALSE;
   S_706.SPARE110 := FALSE;
   S_706.SPARE111 := FALSE;
   S_706.SPARE112 := FALSE;
   S_706.SPARE113 := FALSE;
   S_706.SPARE114 := FALSE;
   S_706.SPARE115 := FALSE;
   S_706.SPARE116 := FALSE;
   S_706.SPARE117 := FALSE;
   S_706.SPARE118 := FALSE;
   S_706.SPARE119 := FALSE;
   S_706.SPARE120 := FALSE;
   S_706.SPARE121 := FALSE;
   S_706.SPARE122 := FALSE;
   S_706.SPARE123 := FALSE;
   S_706.SPARE124 := FALSE;
   S_706.SPARE125 := FALSE;
   S_706.SPARE126 := FALSE;
   S_706.SPARE127 := FALSE;
   S_706.SPARE128 := FALSE;
   S_706.SPARE129 := FALSE;
   S_706.SPARE130 := FALSE;
   S_706.SPARE131 := FALSE;
   S_706.SPARE132 := FALSE;
   S_706.SPARE133 := FALSE;
   S_706.SPARE134 := FALSE;
   S_706.SPARE135 := FALSE;
   S_706.SPARE136 := FALSE;
   S_706.SPARE137 := FALSE;
   S_706.SPARE138 := FALSE;
   S_706.SPARE139 := FALSE;
   S_706.SPARE140 := FALSE;
   S_706.SPARE141 := FALSE;
   S_706.SPARE142 := FALSE;
   S_706.SPARE143 := FALSE;
   S_706.SPARE144 := FALSE;
   S_706.SPARE145 := FALSE;
   S_706.SPARE146 := FALSE;
   S_706.SPARE147 := FALSE;
   S_706.SPARE148 := FALSE;
   S_706.SPARE149 := FALSE;
   S_706.SPARE150 := FALSE;
   S_706.SPARE151 := FALSE;
   S_706.SPARE152 := FALSE;
   S_706.SPARE153 := FALSE;
   S_706.SPARE154 := FALSE;
   S_706.SPARE155 := FALSE;
   S_706.SPARE156 := FALSE;
   S_706.SPARE157 := FALSE;
   S_706.SPARE158 := FALSE;
   S_706.SPARE159 := FALSE;
   S_706.SPARE160 := FALSE;
   S_706.SPARE161 := FALSE;
   S_706.HOOK_PIN_UP_LP := W#16#0;
   S_706.HOOK_PIN_DOWN_LP := W#16#300;
   S_706.DAECHA_LOCK_ADV_LP := W#16#300;
   S_706.DAECHA_LOCK_RET_LP := W#16#0;
   S_706.ELE_ADV_LP := W#16#300;
   S_706.ELE_RET_LP := W#16#0;
   S_706.AIR_ELE_ADV_LP := W#16#300;
   S_706.AIR_ELE_RET_LP := W#16#0;
   S_706.SP_WORD19 := W#16#0;
   S_706.SP_WORD20 := W#16#0;
   S_706.LM_DC_PIN_UP_LP := W#16#0;
   S_706.LM_DC_PIN_DOWN_LP := W#16#0;
   S_706.LM_DC_1ST_CLAMP1_ADV_LP := W#16#0;
   S_706.LM_DC_1ST_CLAMP1_RET_LP := W#16#0;
   S_706.LM_DC_1ST_CLAMP2_ADV_LP := W#16#0;
   S_706.LM_DC_1ST_CLAMP2_RET_LP := W#16#0;
   S_706.LM_DC_1ST_CLAMP3_ADV_LP := W#16#0;
   S_706.LM_DC_1ST_CLAMP3_RET_LP := W#16#0;
   S_706.LM_DC_1ST_CLAMP4_ADV_LP := W#16#0;
   S_706.LM_DC_1ST_CLAMP4_RET_LP := W#16#0;
   S_706.LM_DC_2ND_CLAMP1_ADV_LP := W#16#0;
   S_706.LM_DC_2ND_CLAMP1_RET_LP := W#16#0;
   S_706.LM_DC_2ND_CLAMP2_ADV_LP := W#16#0;
   S_706.LM_DC_2ND_CLAMP2_RET_LP := W#16#0;
   S_706.LM_DC_2ND_CLAMP3_ADV_LP := W#16#0;
   S_706.LM_DC_2ND_CLAMP3_RET_LP := W#16#0;
   S_706.LM_DC_2ND_CLAMP4_ADV_LP := W#16#0;
   S_706.LM_DC_2ND_CLAMP4_RET_LP := W#16#0;
   S_706.LM_DC_2ND_CLAMP5_ADV_LP := W#16#0;
   S_706.LM_DC_2ND_CLAMP5_RET_LP := W#16#0;
   S_706.LM_DC_DR_STK_PIN_UP_LP := W#16#0;
   S_706.LM_DC_DR_STK_PIN_DOWN_LP := W#16#0;
   S_706.LM_DC_OTR_CLAMP_ADV_LP := W#16#0;
   S_706.LM_DC_OTR_CLAMP_RET_LP := W#16#0;
   S_706.LM_DC_ASSY_CLAMP_ADV_LP := W#16#0;
   S_706.LM_DC_ASSY_CLAMP_RET_LP := W#16#0;
   S_706.LM_DC_FF_PIN_UP_LP := W#16#0;
   S_706.LM_DC_FF_PIN_DOWN_LP := W#16#0;
   S_706.LM_DC_FF_CLAMP_ADV_LP := W#16#0;
   S_706.LM_DC_FF_CLAMP_RET_LP := W#16#0;
   S_706.LM_DC_2ND_CLAMP6_ADV_LP := W#16#0;
   S_706.LM_DC_2ND_CLAMP6_RET_LP := W#16#0;
   S_706.LM_DC_2ND_CLAMP7_ADV_LP := W#16#0;
   S_706.LM_DC_2ND_CLAMP7_RET_LP := W#16#0;
   S_706.LM_DC_1ST_CLAMP5_ADV_LP := W#16#0;
   S_706.LM_DC_1ST_CLAMP5_RET_LP := W#16#0;
   S_706.SP_WORD68 := W#16#0;
   S_706.SP_WORD69 := W#16#0;
   S_706.SP_WORD70 := W#16#0;
   S_706.SP_WORD71 := W#16#0;
   S_706.TL_DC_PIN_UP_LP := W#16#F00;
   S_706.TL_DC_PIN_DOWN_LP := W#16#0;
   S_706.TL_DC_LATCH1_ADV_LP := W#16#3F00;
   S_706.TL_DC_LATCH1_RET_LP := W#16#0;
   S_706.TL_DC_LATCH2_ADV_LP := W#16#700;
   S_706.TL_DC_LATCH2_RET_LP := W#16#0;
   S_706.TL_DC_1ST_CLAMP1_ADV_LP := W#16#300;
   S_706.TL_DC_1ST_CLAMP1_RET_LP := W#16#0;
   S_706.TL_DC_1ST_CLAMP2_ADV_LP := W#16#300;
   S_706.TL_DC_1ST_CLAMP2_RET_LP := W#16#0;
   S_706.TL_DC_1ST_CLAMP3_ADV_LP := W#16#300;
   S_706.TL_DC_1ST_CLAMP3_RET_LP := W#16#0;
   S_706.TL_DC_2ND_CLAMP1_ADV_LP := W#16#300;
   S_706.TL_DC_2ND_CLAMP1_RET_LP := W#16#0;
   S_706.TL_DC_2ND_CLAMP2_ADV_LP := W#16#300;
   S_706.TL_DC_2ND_CLAMP2_RET_LP := W#16#0;
   S_706.TL_DC_U261_ADV_LP := W#16#300;
   S_706.TL_DC_U261_RET_LP := W#16#0;
   S_706.TL_DC_U261_CLAMP_ADV_LP := W#16#100;
   S_706.TL_DC_U261_CLAMP_RET_LP := W#16#0;
   S_706.TL_DC_U269_UP_LP := W#16#300;
   S_706.TL_DC_U269_DOWN_LP := W#16#0;
   S_706.TL_DC_U269_CLAMP_ADV_LP := W#16#300;
   S_706.TL_DC_U269_CLAMP_RET_LP := W#16#0;
   S_706.TL_DC_3RD_CLAMP_ADV_LP := W#16#300;
   S_706.TL_DC_3RD_CLAMP_RET_LP := W#16#0;
   S_706.TL_DC_U262_1_UP_LP := W#16#0;
   S_706.TL_DC_U262_1_DOWN_LP := W#16#300;
   S_706.TL_DC_U262_1_ADV_LP := W#16#0;
   S_706.TL_DC_U262_1_RET_LP := W#16#300;
   S_706.TL_DC_U262_1_CLP_ADV_LP := W#16#0;
   S_706.TL_DC_U262_1_CLP_RET_LP := W#16#300;
   S_706.TL_DC_U261_2_CLP_ADV_LP := W#16#0;
   S_706.TL_DC_U261_2_CLP_RET_LP := W#16#300;
   S_706.SP_WORD106 := W#16#0;
   S_706.SP_WORD107 := W#16#0;
   S_706.SP_WORD108 := W#16#0;
   S_706.SP_WORD109 := W#16#0;
   S_706.SP_WORD110 := W#16#0;
   S_706.SP_WORD111 := W#16#0;
   S_707.M_AUTO_SEL := FALSE;
   S_707.M_MANUAL_SEL := FALSE;
   S_707.M_READY_PB := FALSE;
   S_707.M_AUTO_RUN_PB := FALSE;
   S_707.M_WORK_COMP_SET_PB := FALSE;
   S_707.M_WORK_COMP_RST_PB := FALSE;
   S_707.M_HOME_POS_PB := FALSE;
   S_707.M_TIP_DRESS_PB := FALSE;
   S_707.HOOK_PIN_SEL := FALSE;
   S_707.DAECHA_LOCK_SEL := FALSE;
   S_707.ELE_SEL := FALSE;
   S_707.SPARE12 := FALSE;
   S_707.SPARE13 := FALSE;
   S_707.SPARE14 := FALSE;
   S_707.SPARE15 := FALSE;
   S_707.SPARE16 := FALSE;
   S_707.SPARE17 := FALSE;
   S_707.SPARE18 := FALSE;
   S_707.SPARE19 := FALSE;
   S_707.SPARE20 := FALSE;
   S_707.SPARE21 := FALSE;
   S_707.SPARE22 := FALSE;
   S_707.SPARE23 := FALSE;
   S_707.SPARE24 := FALSE;
   S_707.SPARE25 := FALSE;
   S_707.SPARE26 := FALSE;
   S_707.SPARE27 := FALSE;
   S_707.SPARE28 := FALSE;
   S_707.SPARE29 := FALSE;
   S_707.SPARE30 := FALSE;
   S_707.M_ADV_PB := FALSE;
   S_707.M_RET_PB := FALSE;
   S_707.LM_DC_PIN_SEL := FALSE;
   S_707.LM_DC_1ST_CLAMP1_SEL := FALSE;
   S_707.LM_DC_1ST_CLAMP2_SEL := FALSE;
   S_707.LM_DC_1ST_CLAMP3_SEL := FALSE;
   S_707.LM_DC_1ST_CLAMP4_SEL := FALSE;
   S_707.LM_DC_2ND_CLAMP1_SEL := FALSE;
   S_707.LM_DC_2ND_CLAMP2_SEL := FALSE;
   S_707.LM_DC_2ND_CLAMP3_SEL := FALSE;
   S_707.LM_DC_2ND_CLAMP4_SEL := FALSE;
   S_707.LM_DC_2ND_CLAMP5_SEL := FALSE;
   S_707.LM_DC_DR_STK_PIN_SEL := FALSE;
   S_707.LM_DC_OTR_CLAMP_SEL := FALSE;
   S_707.LM_DC_ASSY_CLAMP_SEL := FALSE;
   S_707.LM_DC_FF_PIN_SEL := FALSE;
   S_707.LM_DC_FF_CLAMP_SEL := FALSE;
   S_707.LM_DC_2ND_CLAMP6_SEL := FALSE;
   S_707.SPARE50 := FALSE;
   S_707.SPARE51 := FALSE;
   S_707.SPARE52 := FALSE;
   S_707.SPARE53 := FALSE;
   S_707.SPARE54 := FALSE;
   S_707.SPARE55 := FALSE;
   S_707.SPARE56 := FALSE;
   S_707.SPARE57 := FALSE;
   S_707.SPARE58 := FALSE;
   S_707.SPARE59 := FALSE;
   S_707.SPARE60 := FALSE;
   S_707.SPARE61 := FALSE;
   S_707.SPARE62 := FALSE;
   S_707.SPARE63 := FALSE;
   S_707.LM_DC_M_ADV_PB := FALSE;
   S_707.LM_DC_M_RET_PB := FALSE;
   S_707.TL_DC_PIN_SEL := FALSE;
   S_707.TL_DC_LATCH1_SEL := FALSE;
   S_707.TL_DC_1ST_CLAMP_SEL := FALSE;
   S_707.TL_DC_2ND_CLAMP_SEL := FALSE;
   S_707.TL_DC_U261_SEL := FALSE;
   S_707.TL_DC_U261_CLAMP_SEL := FALSE;
   S_707.TL_DC_U269_UP_DN_SEL := FALSE;
   S_707.TL_DC_U269_CLAMP_SEL := FALSE;
   S_707.TL_DC_3RD_CLAMP_SEL := FALSE;
   S_707.TL_DC_U262_1_UP_DN_SEL := FALSE;
   S_707.TL_DC_U262_1_SEL := FALSE;
   S_707.TL_DC_U262_1_CLAMP_SEL := FALSE;
   S_707.TL_DC_U261_2_CLAMP_SEL := FALSE;
   S_707.SPARE79 := FALSE;
   S_707.SPARE80 := FALSE;
   S_707.SPARE81 := FALSE;
   S_707.SPARE82 := FALSE;
   S_707.SPARE83 := FALSE;
   S_707.SPARE84 := FALSE;
   S_707.SPARE85 := FALSE;
   S_707.SPARE86 := FALSE;
   S_707.SPARE87 := FALSE;
   S_707.SPARE88 := FALSE;
